gfCNCPoint1[12076] = {X 239.3673, Y 29.5319, Z -1.3333, A 0.000, B 0.000, C 0.000 }
gfCNCPoint1[12077] = {X 238.5512, Y 28.3732, Z -1.3333, A 0.000, B 0.000, C 0.000 }
gfCNCPoint1[12078] = {X 237.8897, Y 27.1197, Z -1.3333, A 0.000, B 0.000, C 0.000 }
gfCNCPoint1[12079] = {X 237.3937, Y 25.7920, Z -1.3333, A 0.000, B 0.000, C 0.000 }
gfCNCPoint1[12080] = {X 236.9799, Y 24.0072, Z -1.3333, A 0.000, B 0.000, C 0.000 }
gfCNCPoint1[12081] = {X 236.7691, Y 22.1872, Z -1.3333, A 0.000, B 0.000, C 0.000 }
gfCNCPoint1[12082] = {X 236.7640, Y 20.3550, Z -1.3333, A 0.000, B 0.000, C 0.000 }
gfCNCPoint1[12083] = {X 236.9646, Y 18.5339, Z -1.3333, A 0.000, B 0.000, C 0.000 }
gfCNCPoint1[12084] = {X 237.3683, Y 16.7468, Z -1.3333, A 0.000, B 0.000, C 0.000 }
gfCNCPoint1[12085] = {X 237.9270, Y 15.2029, Z -1.3333, A 0.000, B 0.000, C 0.000 }
gfCNCPoint1[12086] = {X 238.6980, Y 13.7534, Z -1.3333, A 0.000, B 0.000, C 0.000 }
gfCNCPoint1[12087] = {X 239.6659, Y 12.4272, Z -1.3333, A 0.000, B 0.000, C 0.000 }
gfCNCPoint1[12088] = {X 240.8112, Y 11.2509, Z -1.3333, A 0.000, B 0.000, C 0.000 }
gfCNCPoint1[12089] = {X 242.1110, Y 10.2479, Z -1.3333, A 0.000, B 0.000, C 0.000 }
gfCNCPoint1[12090] = {X 243.5394, Y 9.4385, Z -1.3333, A 0.000, B 0.000, C 0.000 }
gfCNCPoint1[12091] = {X 245.0677, Y 8.8387, Z -1.3333, A 0.000, B 0.000, C 0.000 }
gfCNCPoint1[12092] = {X 246.6654, Y 8.4605, Z -1.3333, A 0.000, B 0.000, C 0.000 }
gfCNCPoint1[12093] = {X 248.7417, Y 8.1916, Z -1.3333, A 0.000, B 0.000, C 0.000 }
gfCNCPoint1[12094] = {X 250.8339, Y 8.1119, Z -1.3333, A 0.000, B 0.000, C 0.000 }
gfCNCPoint1[12095] = {X 266.7614, Y 8.1119, Z -1.3333, A 0.000, B 0.000, C 0.000 }
gfCNCPoint1[12096] = {X 267.6634, Y 8.2203, Z -1.3333, A 0.000, B 0.000, C 0.000 }
gfCNCPoint1[12097] = {X 268.5190, Y 8.5254, Z -1.3333, A 0.000, B 0.000, C 0.000 }
gfCNCPoint1[12098] = {X 269.2860, Y 9.0122, Z -1.3333, A 0.000, B 0.000, C 0.000 }
gfCNCPoint1[12099] = {X 269.9264, Y 9.6566, Z -1.3333, A 0.000, B 0.000, C 0.000 }
gfCNCPoint1[12100] = {X 270.4084, Y 10.4266, Z -1.3333, A 0.000, B 0.000, C 0.000 }
gfCNCPoint1[12101] = {X 270.7082, Y 11.2841, Z -1.3333, A 0.000, B 0.000, C 0.000 }
gfCNCPoint1[12102] = {X 270.8110, Y 12.1867, Z -1.3333, A 0.000, B 0.000, C 0.000 }
gfCNCPoint1[12103] = {X 270.8108, Y 13.0200, Z -1.3333, A 0.000, B 0.000, C 0.000 }
gfCNCPoint1[12104] = {X 270.7022, Y 13.9141, Z -1.3333, A 0.000, B 0.000, C 0.000 }
gfCNCPoint1[12105] = {X 270.4001, Y 14.7626, Z -1.3333, A 0.000, B 0.000, C 0.000 }
gfCNCPoint1[12106] = {X 269.9191, Y 15.5241, Z -1.3333, A 0.000, B 0.000, C 0.000 }
gfCNCPoint1[12107] = {X 269.2828, Y 16.1615, Z -1.3333, A 0.000, B 0.000, C 0.000 }
gfCNCPoint1[12108] = {X 269.2827, Y 28.5937, Z -1.3333, A 0.000, B 0.000, C 0.000 }
gfCNCPoint1[12109] = {X 273.2827, Y 28.5937, Z -1.3333, A 0.000, B 0.000, C 0.000 }
gfCNCPoint1[12110] = {X 269.2027, Y 28.5937, Z -1.3333, A 0.000, B 0.000, C 0.000 }
gfCNCPoint1[12111] = {X 269.2026, Y 41.0663, Z -1.3333, A 0.000, B 0.000, C 0.000 }
gfCNCPoint1[12112] = {X 269.3416, Y 41.1781, Z -1.3333, A 0.000, B 0.000, C 0.000 }
gfCNCPoint1[12113] = {X 269.9279, Y 41.8047, Z -1.3333, A 0.000, B 0.000, C 0.000 }
gfCNCPoint1[12114] = {X 270.3671, Y 42.5419, Z -1.3333, A 0.000, B 0.000, C 0.000 }
gfCNCPoint1[12115] = {X 270.6390, Y 43.3558, Z -1.3333, A 0.000, B 0.000, C 0.000 }
gfCNCPoint1[12116] = {X 270.7310, Y 44.2089, Z -1.3333, A 0.000, B 0.000, C 0.000 }
gfCNCPoint1[12117] = {X 270.7310, Y 45.0000, Z -1.3333, A 0.000, B 0.000, C 0.000 }
gfCNCPoint1[12118] = {X 270.6307, Y 45.8901, Z -1.3333, A 0.000, B 0.000, C 0.000 }
gfCNCPoint1[12119] = {X 270.3349, Y 46.7355, Z -1.3333, A 0.000, B 0.000, C 0.000 }
gfCNCPoint1[12120] = {X 269.8584, Y 47.4940, Z -1.3333, A 0.000, B 0.000, C 0.000 }
gfCNCPoint1[12121] = {X 269.2250, Y 48.1273, Z -1.3333, A 0.000, B 0.000, C 0.000 }
gfCNCPoint1[12122] = {X 268.4666, Y 48.6039, Z -1.3333, A 0.000, B 0.000, C 0.000 }
gfCNCPoint1[12123] = {X 267.6211, Y 48.8997, Z -1.3333, A 0.000, B 0.000, C 0.000 }
gfCNCPoint1[12124] = {X 266.7310, Y 49.0000, Z -1.3333, A 0.000, B 0.000, C 0.000 }
gfCNCPoint1[12125] = {X 260.2876, Y 49.0000, Z -1.3333, A 0.000, B 0.000, C 0.000 }
gfCNCPoint1[12126] = {X 259.3975, Y 48.8997, Z -1.3333, A 0.000, B 0.000, C 0.000 }
gfCNCPoint1[12127] = {X 258.5520, Y 48.6039, Z -1.3333, A 0.000, B 0.000, C 0.000 }
gfCNCPoint1[12128] = {X 257.7936, Y 48.1273, Z -1.3333, A 0.000, B 0.000, C 0.000 }
gfCNCPoint1[12129] = {X 257.1602, Y 47.4939, Z -1.3333, A 0.000, B 0.000, C 0.000 }
gfCNCPoint1[12130] = {X 256.6837, Y 46.7355, Z -1.3333, A 0.000, B 0.000, C 0.000 }
gfCNCPoint1[12131] = {X 256.3878, Y 45.8900, Z -1.3333, A 0.000, B 0.000, C 0.000 }
gfCNCPoint1[12132] = {X 256.2876, Y 45.0000, Z -1.3333, A 0.000, B 0.000, C 0.000 }
gfCNCPoint1[12133] = {X 256.2879, Y 44.1538, Z -1.3333, A 0.000, B 0.000, C 0.000 }
gfCNCPoint1[12134] = {X 256.3986, Y 43.2730, Z -1.3333, A 0.000, B 0.000, C 0.000 }
gfCNCPoint1[12135] = {X 256.7008, Y 42.4382, Z -1.3333, A 0.000, B 0.000, C 0.000 }
gfCNCPoint1[12136] = {X 257.1796, Y 41.6907, Z -1.3333, A 0.000, B 0.000, C 0.000 }
gfCNCPoint1[12137] = {X 257.8115, Y 41.0672, Z -1.3333, A 0.000, B 0.000, C 0.000 }
gfCNCPoint1[12138] = {X 257.8115, Y 34.1538, Z -1.3333, A 0.000, B 0.000, C 0.000 }
gfCNCPoint1[12139] = {X 254.8153, Y 34.1538, Z -1.3333, A 0.000, B 0.000, C 0.000 }
gfCNCPoint1[12140] = {X 254.5724, Y 34.1511, Z -1.3333, A 0.000, B 0.000, C 0.000 }
gfCNCPoint1[12141] = {X 250.1354, Y 42.7952, Z -1.3333, A 0.000, B 0.000, C 0.000 }
gfCNCPoint1[12142] = {X 250.3285, Y 43.4904, Z -1.3333, A 0.000, B 0.000, C 0.000 }
gfCNCPoint1[12143] = {X 250.3936, Y 44.2089, Z -1.3333, A 0.000, B 0.000, C 0.000 }
gfCNCPoint1[12144] = {X 250.3936, Y 45.0000, Z -1.3333, A 0.000, B 0.000, C 0.000 }
gfCNCPoint1[12145] = {X 250.2933, Y 45.8901, Z -1.3333, A 0.000, B 0.000, C 0.000 }
gfCNCPoint1[12146] = {X 249.9974, Y 46.7355, Z -1.3333, A 0.000, B 0.000, C 0.000 }
gfCNCPoint1[12147] = {X 249.5209, Y 47.4940, Z -1.3333, A 0.000, B 0.000, C 0.000 }
gfCNCPoint1[12148] = {X 248.8875, Y 48.1273, Z -1.3333, A 0.000, B 0.000, C 0.000 }
gfCNCPoint1[12149] = {X 248.1291, Y 48.6039, Z -1.3333, A 0.000, B 0.000, C 0.000 }
gfCNCPoint1[12150] = {X 247.2836, Y 48.8997, Z -1.3333, A 0.000, B 0.000, C 0.000 }
gfCNCPoint1[12151] = {X 246.3936, Y 49.0000, Z -1.3333, A 0.000, B 0.000, C 0.000 }
gfCNCPoint1[12152] = {X 239.8075, Y 49.0000, Z -1.3333, A 0.000, B 0.000, C 0.000 }
gfCNCPoint1[12153] = {X 238.9174, Y 48.8997, Z -1.3333, A 0.000, B 0.000, C 0.000 }
gfCNCPoint1[12154] = {X 238.0720, Y 48.6039, Z -1.3333, A 0.000, B 0.000, C 0.000 }
gfCNCPoint1[12155] = {X 237.3135, Y 48.1273, Z -1.3333, A 0.000, B 0.000, C 0.000 }
gfCNCPoint1[12156] = {X 236.6802, Y 47.4940, Z -1.3333, A 0.000, B 0.000, C 0.000 }
gfCNCPoint1[12157] = {X 236.2036, Y 46.7355, Z -1.3333, A 0.000, B 0.000, C 0.000 }
gfCNCPoint1[12158] = {X 235.9078, Y 45.8901, Z -1.3333, A 0.000, B 0.000, C 0.000 }
gfCNCPoint1[12159] = {X 235.8075, Y 45.0000, Z -1.3333, A 0.000, B 0.000, C 0.000 }
gfCNCPoint1[12160] = {X 235.8079, Y 44.1538, Z -1.3333, A 0.000, B 0.000, C 0.000 }
gfCNCPoint1[12161] = {X 235.9027, Y 43.3414, Z -1.3333, A 0.000, B 0.000, C 0.000 }
gfCNCPoint1[12162] = {X 236.1607, Y 42.5654, Z -1.3333, A 0.000, B 0.000, C 0.000 }
gfCNCPoint1[12163] = {X 236.5712, Y 41.8580, Z -1.3333, A 0.000, B 0.000, C 0.000 }
gfCNCPoint1[12164] = {X 237.1169, Y 41.2489, Z -1.3333, A 0.000, B 0.000, C 0.000 }
gfCNCPoint1[12165] = {X 237.7752, Y 40.7635, Z -1.3333, A 0.000, B 0.000, C 0.000 }
gfCNCPoint1[12166] = {X 238.5184, Y 40.4222, Z -1.3333, A 0.000, B 0.000, C 0.000 }
gfCNCPoint1[12167] = {X 242.7051, Y 32.2271, Z -1.3333, A 0.000, B 0.000, C 0.000 }
gfCNCPoint1[12168] = {X 241.5071, Y 31.4650, Z -1.3333, A 0.000, B 0.000, C 0.000 }
gfCNCPoint1[12169] = {X 240.4173, Y 30.5548, Z -1.3333, A 0.000, B 0.000, C 0.000 }
gfCNCPoint1[12170] = {X 239.4538, Y 29.5118, Z -1.3333, A 0.000, B 0.000, C 0.000 }
gfCNCPoint1[12171] = {X 238.6328, Y 28.3533, Z -1.3333, A 0.000, B 0.000, C 0.000 }
gfCNCPoint1[12172] = {X 237.9679, Y 27.0987, Z -1.3333, A 0.000, B 0.000, C 0.000 }
gfCNCPoint1[12173] = {X 237.4702, Y 25.7689, Z -1.3333, A 0.000, B 0.000, C 0.000 }
gfCNCPoint1[12174] = {X 237.0586, Y 23.9929, Z -1.3333, A 0.000, B 0.000, C 0.000 }
gfCNCPoint1[12175] = {X 236.8490, Y 22.1820, Z -1.3333, A 0.000, B 0.000, C 0.000 }
gfCNCPoint1[12176] = {X 236.8439, Y 20.3590, Z -1.3333, A 0.000, B 0.000, C 0.000 }
gfCNCPoint1[12177] = {X 237.0435, Y 18.5469, Z -1.3333, A 0.000, B 0.000, C 0.000 }
gfCNCPoint1[12178] = {X 237.4452, Y 16.7687, Z -1.3333, A 0.000, B 0.000, C 0.000 }
gfCNCPoint1[12179] = {X 238.0001, Y 15.2355, Z -1.3333, A 0.000, B 0.000, C 0.000 }
gfCNCPoint1[12180] = {X 238.7658, Y 13.7959, Z -1.3333, A 0.000, B 0.000, C 0.000 }
gfCNCPoint1[12181] = {X 239.7270, Y 12.4788, Z -1.3333, A 0.000, B 0.000, C 0.000 }
gfCNCPoint1[12182] = {X 240.8645, Y 11.3105, Z -1.3333, A 0.000, B 0.000, C 0.000 }
gfCNCPoint1[12183] = {X 242.1555, Y 10.3144, Z -1.3333, A 0.000, B 0.000, C 0.000 }
gfCNCPoint1[12184] = {X 243.5741, Y 9.5105, Z -1.3333, A 0.000, B 0.000, C 0.000 }
gfCNCPoint1[12185] = {X 245.0920, Y 8.9149, Z -1.3333, A 0.000, B 0.000, C 0.000 }
gfCNCPoint1[12186] = {X 246.6787, Y 8.5394, Z -1.3333, A 0.000, B 0.000, C 0.000 }
gfCNCPoint1[12187] = {X 248.7483, Y 8.2713, Z -1.3333, A 0.000, B 0.000, C 0.000 }
gfCNCPoint1[12188] = {X 250.8336, Y 8.1919, Z -1.3333, A 0.000, B 0.000, C 0.000 }
gfCNCPoint1[12189] = {X 266.7608, Y 8.1919, Z -1.3333, A 0.000, B 0.000, C 0.000 }
gfCNCPoint1[12190] = {X 267.6450, Y 8.2982, Z -1.3333, A 0.000, B 0.000, C 0.000 }
gfCNCPoint1[12191] = {X 268.4839, Y 8.5973, Z -1.3333, A 0.000, B 0.000, C 0.000 }
gfCNCPoint1[12192] = {X 269.2359, Y 9.0746, Z -1.3333, A 0.000, B 0.000, C 0.000 }
gfCNCPoint1[12193] = {X 269.8637, Y 9.7063, Z -1.3333, A 0.000, B 0.000, C 0.000 }
gfCNCPoint1[12194] = {X 270.3363, Y 10.4612, Z -1.3333, A 0.000, B 0.000, C 0.000 }
gfCNCPoint1[12195] = {X 270.6303, Y 11.3020, Z -1.3333, A 0.000, B 0.000, C 0.000 }
gfCNCPoint1[12196] = {X 270.7310, Y 12.1869, Z -1.3333, A 0.000, B 0.000, C 0.000 }
gfCNCPoint1[12197] = {X 270.7308, Y 13.0192, Z -1.3333, A 0.000, B 0.000, C 0.000 }
gfCNCPoint1[12198] = {X 270.6221, Y 13.9051, Z -1.3333, A 0.000, B 0.000, C 0.000 }
gfCNCPoint1[12199] = {X 270.3197, Y 14.7448, Z -1.3333, A 0.000, B 0.000, C 0.000 }
gfCNCPoint1[12200] = {X 269.8386, Y 15.4965, Z -1.3333, A 0.000, B 0.000, C 0.000 }
gfCNCPoint1[12201] = {X 269.2028, Y 16.1229, Z -1.3333, A 0.000, B 0.000, C 0.000 }
gfCNCPoint1[12202] = {X 269.2027, Y 28.5937, Z -1.3333, A 0.000, B 0.000, C 0.000 }
gfCNCPoint1[12203] = {X 273.2827, Y 28.5937, Z -1.3333, A 0.000, B 0.000, C 0.000 }
gfCNCPoint1[12204] = {X 273.2827, Y 28.5937, Z 1.6667, A 0.000, B 0.000, C 0.000 }
gfCNCPoint1[12205] = {X 273.2827, Y 28.5937, Z 11.0000, A 0.000, B 0.000, C 0.000 }
gfCNCPoint1[12206] = {X 277.7463, Y 28.5933, Z 11.0000, A 0.000, B 0.000, C 0.000 }
gfCNCPoint1[12207] = {X 277.7463, Y 28.5933, Z 1.6667, A 0.000, B 0.000, C 0.000 }
gfCNCPoint1[12208] = {X 277.7463, Y 28.5933, Z -1.3333, A 0.000, B 0.000, C 0.000 }
gfCNCPoint1[12209] = {X 281.8263, Y 28.5932, Z -1.3333, A 0.000, B 0.000, C 0.000 }
gfCNCPoint1[12210] = {X 281.8261, Y 16.2749, Z -1.3333, A 0.000, B 0.000, C 0.000 }
gfCNCPoint1[12211] = {X 281.1872, Y 15.6037, Z -1.3333, A 0.000, B 0.000, C 0.000 }
gfCNCPoint1[12212] = {X 280.7062, Y 14.8118, Z -1.3333, A 0.000, B 0.000, C 0.000 }
gfCNCPoint1[12213] = {X 280.4051, Y 13.9354, Z -1.3333, A 0.000, B 0.000, C 0.000 }
gfCNCPoint1[12214] = {X 280.2978, Y 13.0150, Z -1.3333, A 0.000, B 0.000, C 0.000 }
gfCNCPoint1[12215] = {X 280.2977, Y 12.1868, Z -1.3333, A 0.000, B 0.000, C 0.000 }
gfCNCPoint1[12216] = {X 280.4060, Y 11.2255, Z -1.3333, A 0.000, B 0.000, C 0.000 }
gfCNCPoint1[12217] = {X 280.7255, Y 10.3124, Z -1.3333, A 0.000, B 0.000, C 0.000 }
gfCNCPoint1[12218] = {X 281.2402, Y 9.4933, Z -1.3333, A 0.000, B 0.000, C 0.000 }
gfCNCPoint1[12219] = {X 281.9242, Y 8.8093, Z -1.3333, A 0.000, B 0.000, C 0.000 }
gfCNCPoint1[12220] = {X 282.7433, Y 8.2946, Z -1.3333, A 0.000, B 0.000, C 0.000 }
gfCNCPoint1[12221] = {X 283.6564, Y 7.9751, Z -1.3333, A 0.000, B 0.000, C 0.000 }
gfCNCPoint1[12222] = {X 284.6177, Y 7.8668, Z -1.3333, A 0.000, B 0.000, C 0.000 }
gfCNCPoint1[12223] = {X 291.0611, Y 7.8668, Z -1.3333, A 0.000, B 0.000, C 0.000 }
gfCNCPoint1[12224] = {X 292.0224, Y 7.9751, Z -1.3333, A 0.000, B 0.000, C 0.000 }
gfCNCPoint1[12225] = {X 292.9355, Y 8.2946, Z -1.3333, A 0.000, B 0.000, C 0.000 }
gfCNCPoint1[12226] = {X 293.7546, Y 8.8093, Z -1.3333, A 0.000, B 0.000, C 0.000 }
gfCNCPoint1[12227] = {X 294.4386, Y 9.4933, Z -1.3333, A 0.000, B 0.000, C 0.000 }
gfCNCPoint1[12228] = {X 294.9533, Y 10.3124, Z -1.3333, A 0.000, B 0.000, C 0.000 }
gfCNCPoint1[12229] = {X 295.2728, Y 11.2255, Z -1.3333, A 0.000, B 0.000, C 0.000 }
gfCNCPoint1[12230] = {X 295.3811, Y 12.1868, Z -1.3333, A 0.000, B 0.000, C 0.000 }
gfCNCPoint1[12231] = {X 295.3811, Y 12.9781, Z -1.3333, A 0.000, B 0.000, C 0.000 }
gfCNCPoint1[12232] = {X 295.2797, Y 13.9084, Z -1.3333, A 0.000, B 0.000, C 0.000 }
gfCNCPoint1[12233] = {X 294.9802, Y 14.7950, Z -1.3333, A 0.000, B 0.000, C 0.000 }
gfCNCPoint1[12234] = {X 294.4969, Y 15.5963, Z -1.3333, A 0.000, B 0.000, C 0.000 }
gfCNCPoint1[12235] = {X 293.8524, Y 16.2748, Z -1.3333, A 0.000, B 0.000, C 0.000 }
gfCNCPoint1[12236] = {X 293.8537, Y 22.1965, Z -1.3333, A 0.000, B 0.000, C 0.000 }
gfCNCPoint1[12237] = {X 302.7601, Y 22.1965, Z -1.3333, A 0.000, B 0.000, C 0.000 }
gfCNCPoint1[12238] = {X 302.7648, Y 16.2784, Z -1.3333, A 0.000, B 0.000, C 0.000 }
gfCNCPoint1[12239] = {X 302.1245, Y 15.6073, Z -1.3333, A 0.000, B 0.000, C 0.000 }
gfCNCPoint1[12240] = {X 301.6422, Y 14.8149, Z -1.3333, A 0.000, B 0.000, C 0.000 }
gfCNCPoint1[12241] = {X 301.3402, Y 13.9378, Z -1.3333, A 0.000, B 0.000, C 0.000 }
gfCNCPoint1[12242] = {X 301.2324, Y 13.0165, Z -1.3333, A 0.000, B 0.000, C 0.000 }
gfCNCPoint1[12243] = {X 301.2323, Y 12.1868, Z -1.3333, A 0.000, B 0.000, C 0.000 }
gfCNCPoint1[12244] = {X 301.3406, Y 11.2255, Z -1.3333, A 0.000, B 0.000, C 0.000 }
gfCNCPoint1[12245] = {X 301.6601, Y 10.3124, Z -1.3333, A 0.000, B 0.000, C 0.000 }
gfCNCPoint1[12246] = {X 302.1747, Y 9.4933, Z -1.3333, A 0.000, B 0.000, C 0.000 }
gfCNCPoint1[12247] = {X 302.8588, Y 8.8093, Z -1.3333, A 0.000, B 0.000, C 0.000 }
gfCNCPoint1[12248] = {X 303.6779, Y 8.2946, Z -1.3333, A 0.000, B 0.000, C 0.000 }
gfCNCPoint1[12249] = {X 304.5910, Y 7.9751, Z -1.3333, A 0.000, B 0.000, C 0.000 }
gfCNCPoint1[12250] = {X 305.5523, Y 7.8668, Z -1.3333, A 0.000, B 0.000, C 0.000 }
gfCNCPoint1[12251] = {X 311.9957, Y 7.8668, Z -1.3333, A 0.000, B 0.000, C 0.000 }
gfCNCPoint1[12252] = {X 312.9570, Y 7.9751, Z -1.3333, A 0.000, B 0.000, C 0.000 }
gfCNCPoint1[12253] = {X 313.8701, Y 8.2946, Z -1.3333, A 0.000, B 0.000, C 0.000 }
gfCNCPoint1[12254] = {X 314.6892, Y 8.8093, Z -1.3333, A 0.000, B 0.000, C 0.000 }
gfCNCPoint1[12255] = {X 315.3732, Y 9.4933, Z -1.3333, A 0.000, B 0.000, C 0.000 }
gfCNCPoint1[12256] = {X 315.8879, Y 10.3124, Z -1.3333, A 0.000, B 0.000, C 0.000 }
gfCNCPoint1[12257] = {X 316.2074, Y 11.2255, Z -1.3333, A 0.000, B 0.000, C 0.000 }
gfCNCPoint1[12258] = {X 316.3157, Y 12.1868, Z -1.3333, A 0.000, B 0.000, C 0.000 }
gfCNCPoint1[12259] = {X 316.3157, Y 12.9781, Z -1.3333, A 0.000, B 0.000, C 0.000 }
gfCNCPoint1[12260] = {X 316.2143, Y 13.9085, Z -1.3333, A 0.000, B 0.000, C 0.000 }
gfCNCPoint1[12261] = {X 315.9150, Y 14.7951, Z -1.3333, A 0.000, B 0.000, C 0.000 }
gfCNCPoint1[12262] = {X 315.4317, Y 15.5965, Z -1.3333, A 0.000, B 0.000, C 0.000 }
gfCNCPoint1[12263] = {X 314.7871, Y 16.2750, Z -1.3333, A 0.000, B 0.000, C 0.000 }
gfCNCPoint1[12264] = {X 314.7869, Y 40.9116, Z -1.3333, A 0.000, B 0.000, C 0.000 }
gfCNCPoint1[12265] = {X 315.4259, Y 41.5826, Z -1.3333, A 0.000, B 0.000, C 0.000 }
gfCNCPoint1[12266] = {X 315.9070, Y 42.3746, Z -1.3333, A 0.000, B 0.000, C 0.000 }
gfCNCPoint1[12267] = {X 316.2082, Y 43.2509, Z -1.3333, A 0.000, B 0.000, C 0.000 }
gfCNCPoint1[12268] = {X 316.3156, Y 44.1713, Z -1.3333, A 0.000, B 0.000, C 0.000 }
gfCNCPoint1[12269] = {X 316.3157, Y 45.0000, Z -1.3333, A 0.000, B 0.000, C 0.000 }
gfCNCPoint1[12270] = {X 316.2074, Y 45.9613, Z -1.3333, A 0.000, B 0.000, C 0.000 }
gfCNCPoint1[12271] = {X 315.8879, Y 46.8744, Z -1.3333, A 0.000, B 0.000, C 0.000 }
gfCNCPoint1[12272] = {X 315.3732, Y 47.6935, Z -1.3333, A 0.000, B 0.000, C 0.000 }
gfCNCPoint1[12273] = {X 314.6892, Y 48.3775, Z -1.3333, A 0.000, B 0.000, C 0.000 }
gfCNCPoint1[12274] = {X 313.8701, Y 48.8922, Z -1.3333, A 0.000, B 0.000, C 0.000 }
gfCNCPoint1[12275] = {X 312.9570, Y 49.2117, Z -1.3333, A 0.000, B 0.000, C 0.000 }
gfCNCPoint1[12276] = {X 311.9957, Y 49.3200, Z -1.3333, A 0.000, B 0.000, C 0.000 }
gfCNCPoint1[12277] = {X 305.5523, Y 49.3200, Z -1.3333, A 0.000, B 0.000, C 0.000 }
gfCNCPoint1[12278] = {X 304.5958, Y 49.2128, Z -1.3333, A 0.000, B 0.000, C 0.000 }
gfCNCPoint1[12279] = {X 303.6868, Y 48.8965, Z -1.3333, A 0.000, B 0.000, C 0.000 }
gfCNCPoint1[12280] = {X 302.8704, Y 48.3868, Z -1.3333, A 0.000, B 0.000, C 0.000 }
gfCNCPoint1[12281] = {X 302.1872, Y 47.7090, Z -1.3333, A 0.000, B 0.000, C 0.000 }
gfCNCPoint1[12282] = {X 301.6709, Y 46.8967, Z -1.3333, A 0.000, B 0.000, C 0.000 }
gfCNCPoint1[12283] = {X 301.3473, Y 45.9903, Z -1.3333, A 0.000, B 0.000, C 0.000 }
gfCNCPoint1[12284] = {X 301.2324, Y 45.0348, Z -1.3333, A 0.000, B 0.000, C 0.000 }
gfCNCPoint1[12285] = {X 301.2324, Y 44.2010, Z -1.3333, A 0.000, B 0.000, C 0.000 }
gfCNCPoint1[12286] = {X 301.3506, Y 43.2650, Z -1.3333, A 0.000, B 0.000, C 0.000 }
gfCNCPoint1[12287] = {X 301.6542, Y 42.3717, Z -1.3333, A 0.000, B 0.000, C 0.000 }
gfCNCPoint1[12288] = {X 302.1308, Y 41.5575, Z -1.3333, A 0.000, B 0.000, C 0.000 }
gfCNCPoint1[12289] = {X 302.7611, Y 40.8554, Z -1.3333, A 0.000, B 0.000, C 0.000 }
gfCNCPoint1[12290] = {X 302.7611, Y 34.0343, Z -1.3333, A 0.000, B 0.000, C 0.000 }
gfCNCPoint1[12291] = {X 293.8535, Y 34.0343, Z -1.3333, A 0.000, B 0.000, C 0.000 }
gfCNCPoint1[12292] = {X 293.8525, Y 40.9029, Z -1.3333, A 0.000, B 0.000, C 0.000 }
gfCNCPoint1[12293] = {X 294.4915, Y 41.5869, Z -1.3333, A 0.000, B 0.000, C 0.000 }
gfCNCPoint1[12294] = {X 294.9723, Y 42.3901, Z -1.3333, A 0.000, B 0.000, C 0.000 }
gfCNCPoint1[12295] = {X 295.2733, Y 43.2764, Z -1.3333, A 0.000, B 0.000, C 0.000 }
gfCNCPoint1[12296] = {X 295.3811, Y 44.2063, Z -1.3333, A 0.000, B 0.000, C 0.000 }
gfCNCPoint1[12297] = {X 295.3811, Y 45.0000, Z -1.3333, A 0.000, B 0.000, C 0.000 }
gfCNCPoint1[12298] = {X 295.2728, Y 45.9613, Z -1.3333, A 0.000, B 0.000, C 0.000 }
gfCNCPoint1[12299] = {X 294.9533, Y 46.8744, Z -1.3333, A 0.000, B 0.000, C 0.000 }
gfCNCPoint1[12300] = {X 294.4386, Y 47.6935, Z -1.3333, A 0.000, B 0.000, C 0.000 }
gfCNCPoint1[12301] = {X 293.7546, Y 48.3775, Z -1.3333, A 0.000, B 0.000, C 0.000 }
gfCNCPoint1[12302] = {X 292.9355, Y 48.8922, Z -1.3333, A 0.000, B 0.000, C 0.000 }
gfCNCPoint1[12303] = {X 292.0224, Y 49.2117, Z -1.3333, A 0.000, B 0.000, C 0.000 }
gfCNCPoint1[12304] = {X 291.0611, Y 49.3200, Z -1.3333, A 0.000, B 0.000, C 0.000 }
gfCNCPoint1[12305] = {X 284.6177, Y 49.3200, Z -1.3333, A 0.000, B 0.000, C 0.000 }
gfCNCPoint1[12306] = {X 283.6613, Y 49.2128, Z -1.3333, A 0.000, B 0.000, C 0.000 }
gfCNCPoint1[12307] = {X 282.7524, Y 48.8965, Z -1.3333, A 0.000, B 0.000, C 0.000 }
gfCNCPoint1[12308] = {X 281.9360, Y 48.3869, Z -1.3333, A 0.000, B 0.000, C 0.000 }
gfCNCPoint1[12309] = {X 281.2527, Y 47.7092, Z -1.3333, A 0.000, B 0.000, C 0.000 }
gfCNCPoint1[12310] = {X 280.7365, Y 46.8970, Z -1.3333, A 0.000, B 0.000, C 0.000 }
gfCNCPoint1[12311] = {X 280.4128, Y 45.9907, Z -1.3333, A 0.000, B 0.000, C 0.000 }
gfCNCPoint1[12312] = {X 280.2978, Y 45.0352, Z -1.3333, A 0.000, B 0.000, C 0.000 }
gfCNCPoint1[12313] = {X 280.2977, Y 44.2069, Z -1.3333, A 0.000, B 0.000, C 0.000 }
gfCNCPoint1[12314] = {X 280.4033, Y 43.2781, Z -1.3333, A 0.000, B 0.000, C 0.000 }
gfCNCPoint1[12315] = {X 280.7038, Y 42.3930, Z -1.3333, A 0.000, B 0.000, C 0.000 }
gfCNCPoint1[12316] = {X 281.1856, Y 41.5919, Z -1.3333, A 0.000, B 0.000, C 0.000 }
gfCNCPoint1[12317] = {X 281.8265, Y 40.9115, Z -1.3333, A 0.000, B 0.000, C 0.000 }
gfCNCPoint1[12318] = {X 281.8263, Y 28.5932, Z -1.3333, A 0.000, B 0.000, C 0.000 }
gfCNCPoint1[12319] = {X 277.8263, Y 28.5933, Z -1.3333, A 0.000, B 0.000, C 0.000 }
gfCNCPoint1[12320] = {X 281.9063, Y 28.5932, Z -1.3333, A 0.000, B 0.000, C 0.000 }
gfCNCPoint1[12321] = {X 281.9061, Y 16.2376, Z -1.3333, A 0.000, B 0.000, C 0.000 }
gfCNCPoint1[12322] = {X 281.2677, Y 15.5771, Z -1.3333, A 0.000, B 0.000, C 0.000 }
gfCNCPoint1[12323] = {X 280.7865, Y 14.7945, Z -1.3333, A 0.000, B 0.000, C 0.000 }
gfCNCPoint1[12324] = {X 280.4852, Y 13.9267, Z -1.3333, A 0.000, B 0.000, C 0.000 }
gfCNCPoint1[12325] = {X 280.3778, Y 13.0143, Z -1.3333, A 0.000, B 0.000, C 0.000 }
gfCNCPoint1[12326] = {X 280.3777, Y 12.1868, Z -1.3333, A 0.000, B 0.000, C 0.000 }
gfCNCPoint1[12327] = {X 280.4840, Y 11.2433, Z -1.3333, A 0.000, B 0.000, C 0.000 }
gfCNCPoint1[12328] = {X 280.7976, Y 10.3472, Z -1.3333, A 0.000, B 0.000, C 0.000 }
gfCNCPoint1[12329] = {X 281.3027, Y 9.5432, Z -1.3333, A 0.000, B 0.000, C 0.000 }
gfCNCPoint1[12330] = {X 281.9741, Y 8.8719, Z -1.3333, A 0.000, B 0.000, C 0.000 }
gfCNCPoint1[12331] = {X 282.7780, Y 8.3667, Z -1.3333, A 0.000, B 0.000, C 0.000 }
gfCNCPoint1[12332] = {X 283.6742, Y 8.0531, Z -1.3333, A 0.000, B 0.000, C 0.000 }
gfCNCPoint1[12333] = {X 284.6177, Y 7.9468, Z -1.3333, A 0.000, B 0.000, C 0.000 }
gfCNCPoint1[12334] = {X 291.0611, Y 7.9468, Z -1.3333, A 0.000, B 0.000, C 0.000 }
gfCNCPoint1[12335] = {X 292.0046, Y 8.0531, Z -1.3333, A 0.000, B 0.000, C 0.000 }
gfCNCPoint1[12336] = {X 292.9008, Y 8.3667, Z -1.3333, A 0.000, B 0.000, C 0.000 }
gfCNCPoint1[12337] = {X 293.7047, Y 8.8718, Z -1.3333, A 0.000, B 0.000, C 0.000 }
gfCNCPoint1[12338] = {X 294.3761, Y 9.5432, Z -1.3333, A 0.000, B 0.000, C 0.000 }
gfCNCPoint1[12339] = {X 294.8812, Y 10.3471, Z -1.3333, A 0.000, B 0.000, C 0.000 }
gfCNCPoint1[12340] = {X 295.1948, Y 11.2433, Z -1.3333, A 0.000, B 0.000, C 0.000 }
gfCNCPoint1[12341] = {X 295.3011, Y 12.1868, Z -1.3333, A 0.000, B 0.000, C 0.000 }
gfCNCPoint1[12342] = {X 295.3011, Y 12.9781, Z -1.3333, A 0.000, B 0.000, C 0.000 }
gfCNCPoint1[12343] = {X 295.1995, Y 13.9002, Z -1.3333, A 0.000, B 0.000, C 0.000 }
gfCNCPoint1[12344] = {X 294.8999, Y 14.7781, Z -1.3333, A 0.000, B 0.000, C 0.000 }
gfCNCPoint1[12345] = {X 294.4164, Y 15.5698, Z -1.3333, A 0.000, B 0.000, C 0.000 }
gfCNCPoint1[12346] = {X 293.7724, Y 16.2375, Z -1.3333, A 0.000, B 0.000, C 0.000 }
gfCNCPoint1[12347] = {X 293.7738, Y 22.2765, Z -1.3333, A 0.000, B 0.000, C 0.000 }
gfCNCPoint1[12348] = {X 302.8400, Y 22.2765, Z -1.3333, A 0.000, B 0.000, C 0.000 }
gfCNCPoint1[12349] = {X 302.8449, Y 16.2411, Z -1.3333, A 0.000, B 0.000, C 0.000 }
gfCNCPoint1[12350] = {X 302.2050, Y 15.5806, Z -1.3333, A 0.000, B 0.000, C 0.000 }
gfCNCPoint1[12351] = {X 301.7226, Y 14.7976, Z -1.3333, A 0.000, B 0.000, C 0.000 }
gfCNCPoint1[12352] = {X 301.4203, Y 13.9291, Z -1.3333, A 0.000, B 0.000, C 0.000 }
gfCNCPoint1[12353] = {X 301.3124, Y 13.0158, Z -1.3333, A 0.000, B 0.000, C 0.000 }
gfCNCPoint1[12354] = {X 301.3123, Y 12.1868, Z -1.3333, A 0.000, B 0.000, C 0.000 }
gfCNCPoint1[12355] = {X 301.4186, Y 11.2433, Z -1.3333, A 0.000, B 0.000, C 0.000 }
gfCNCPoint1[12356] = {X 301.7321, Y 10.3471, Z -1.3333, A 0.000, B 0.000, C 0.000 }
gfCNCPoint1[12357] = {X 302.2373, Y 9.5432, Z -1.3333, A 0.000, B 0.000, C 0.000 }
gfCNCPoint1[12358] = {X 302.9087, Y 8.8718, Z -1.3333, A 0.000, B 0.000, C 0.000 }
gfCNCPoint1[12359] = {X 303.7126, Y 8.3667, Z -1.3333, A 0.000, B 0.000, C 0.000 }
gfCNCPoint1[12360] = {X 304.6088, Y 8.0531, Z -1.3333, A 0.000, B 0.000, C 0.000 }
gfCNCPoint1[12361] = {X 305.5523, Y 7.9468, Z -1.3333, A 0.000, B 0.000, C 0.000 }
gfCNCPoint1[12362] = {X 311.9957, Y 7.9468, Z -1.3333, A 0.000, B 0.000, C 0.000 }
gfCNCPoint1[12363] = {X 312.9392, Y 8.0531, Z -1.3333, A 0.000, B 0.000, C 0.000 }
gfCNCPoint1[12364] = {X 313.8354, Y 8.3667, Z -1.3333, A 0.000, B 0.000, C 0.000 }
gfCNCPoint1[12365] = {X 314.6393, Y 8.8718, Z -1.3333, A 0.000, B 0.000, C 0.000 }
gfCNCPoint1[12366] = {X 315.3107, Y 9.5432, Z -1.3333, A 0.000, B 0.000, C 0.000 }
gfCNCPoint1[12367] = {X 315.8158, Y 10.3471, Z -1.3333, A 0.000, B 0.000, C 0.000 }
gfCNCPoint1[12368] = {X 316.1294, Y 11.2433, Z -1.3333, A 0.000, B 0.000, C 0.000 }
gfCNCPoint1[12369] = {X 316.2357, Y 12.1868, Z -1.3333, A 0.000, B 0.000, C 0.000 }
gfCNCPoint1[12370] = {X 316.2357, Y 12.9781, Z -1.3333, A 0.000, B 0.000, C 0.000 }
gfCNCPoint1[12371] = {X 316.1342, Y 13.9003, Z -1.3333, A 0.000, B 0.000, C 0.000 }
gfCNCPoint1[12372] = {X 315.8346, Y 14.7782, Z -1.3333, A 0.000, B 0.000, C 0.000 }
gfCNCPoint1[12373] = {X 315.3512, Y 15.5700, Z -1.3333, A 0.000, B 0.000, C 0.000 }
gfCNCPoint1[12374] = {X 314.7071, Y 16.2377, Z -1.3333, A 0.000, B 0.000, C 0.000 }
gfCNCPoint1[12375] = {X 314.7069, Y 40.9503, Z -1.3333, A 0.000, B 0.000, C 0.000 }
gfCNCPoint1[12376] = {X 314.7352, Y 40.9726, Z -1.3333, A 0.000, B 0.000, C 0.000 }
gfCNCPoint1[12377] = {X 315.3623, Y 41.6313, Z -1.3333, A 0.000, B 0.000, C 0.000 }
gfCNCPoint1[12378] = {X 315.8346, Y 42.4085, Z -1.3333, A 0.000, B 0.000, C 0.000 }
gfCNCPoint1[12379] = {X 316.1302, Y 43.2686, Z -1.3333, A 0.000, B 0.000, C 0.000 }
gfCNCPoint1[12380] = {X 316.2356, Y 44.1720, Z -1.3333, A 0.000, B 0.000, C 0.000 }
gfCNCPoint1[12381] = {X 316.2357, Y 45.0000, Z -1.3333, A 0.000, B 0.000, C 0.000 }
gfCNCPoint1[12382] = {X 316.1294, Y 45.9435, Z -1.3333, A 0.000, B 0.000, C 0.000 }
gfCNCPoint1[12383] = {X 315.8158, Y 46.8397, Z -1.3333, A 0.000, B 0.000, C 0.000 }
gfCNCPoint1[12384] = {X 315.3107, Y 47.6436, Z -1.3333, A 0.000, B 0.000, C 0.000 }
gfCNCPoint1[12385] = {X 314.6393, Y 48.3150, Z -1.3333, A 0.000, B 0.000, C 0.000 }
gfCNCPoint1[12386] = {X 313.8354, Y 48.8201, Z -1.3333, A 0.000, B 0.000, C 0.000 }
gfCNCPoint1[12387] = {X 312.9392, Y 49.1337, Z -1.3333, A 0.000, B 0.000, C 0.000 }
gfCNCPoint1[12388] = {X 311.9957, Y 49.2400, Z -1.3333, A 0.000, B 0.000, C 0.000 }
gfCNCPoint1[12389] = {X 305.5523, Y 49.2400, Z -1.3333, A 0.000, B 0.000, C 0.000 }
gfCNCPoint1[12390] = {X 304.6135, Y 49.1348, Z -1.3333, A 0.000, B 0.000, C 0.000 }
gfCNCPoint1[12391] = {X 303.7214, Y 48.8243, Z -1.3333, A 0.000, B 0.000, C 0.000 }
gfCNCPoint1[12392] = {X 302.9201, Y 48.3241, Z -1.3333, A 0.000, B 0.000, C 0.000 }
gfCNCPoint1[12393] = {X 302.2495, Y 47.6588, Z -1.3333, A 0.000, B 0.000, C 0.000 }
gfCNCPoint1[12394] = {X 301.7428, Y 46.8616, Z -1.3333, A 0.000, B 0.000, C 0.000 }
gfCNCPoint1[12395] = {X 301.4252, Y 45.9720, Z -1.3333, A 0.000, B 0.000, C 0.000 }
gfCNCPoint1[12396] = {X 301.3124, Y 45.0341, Z -1.3333, A 0.000, B 0.000, C 0.000 }
gfCNCPoint1[12397] = {X 301.3123, Y 44.2030, Z -1.3333, A 0.000, B 0.000, C 0.000 }
gfCNCPoint1[12398] = {X 301.4305, Y 43.2744, Z -1.3333, A 0.000, B 0.000, C 0.000 }
gfCNCPoint1[12399] = {X 301.7343, Y 42.3889, Z -1.3333, A 0.000, B 0.000, C 0.000 }
gfCNCPoint1[12400] = {X 302.2111, Y 41.5833, Z -1.3333, A 0.000, B 0.000, C 0.000 }
gfCNCPoint1[12401] = {X 302.8411, Y 40.8909, Z -1.3333, A 0.000, B 0.000, C 0.000 }
gfCNCPoint1[12402] = {X 302.8411, Y 33.9543, Z -1.3333, A 0.000, B 0.000, C 0.000 }
gfCNCPoint1[12403] = {X 293.7735, Y 33.9543, Z -1.3333, A 0.000, B 0.000, C 0.000 }
gfCNCPoint1[12404] = {X 293.7724, Y 40.9397, Z -1.3333, A 0.000, B 0.000, C 0.000 }
gfCNCPoint1[12405] = {X 294.4111, Y 41.6133, Z -1.3333, A 0.000, B 0.000, C 0.000 }
gfCNCPoint1[12406] = {X 294.8920, Y 42.4072, Z -1.3333, A 0.000, B 0.000, C 0.000 }
gfCNCPoint1[12407] = {X 295.1933, Y 43.2851, Z -1.3333, A 0.000, B 0.000, C 0.000 }
gfCNCPoint1[12408] = {X 295.3011, Y 44.2070, Z -1.3333, A 0.000, B 0.000, C 0.000 }
gfCNCPoint1[12409] = {X 295.3011, Y 45.0000, Z -1.3333, A 0.000, B 0.000, C 0.000 }
gfCNCPoint1[12410] = {X 295.1948, Y 45.9435, Z -1.3333, A 0.000, B 0.000, C 0.000 }
gfCNCPoint1[12411] = {X 294.8812, Y 46.8397, Z -1.3333, A 0.000, B 0.000, C 0.000 }
gfCNCPoint1[12412] = {X 294.3761, Y 47.6436, Z -1.3333, A 0.000, B 0.000, C 0.000 }
gfCNCPoint1[12413] = {X 293.7047, Y 48.3150, Z -1.3333, A 0.000, B 0.000, C 0.000 }
gfCNCPoint1[12414] = {X 292.9008, Y 48.8201, Z -1.3333, A 0.000, B 0.000, C 0.000 }
gfCNCPoint1[12415] = {X 292.0046, Y 49.1337, Z -1.3333, A 0.000, B 0.000, C 0.000 }
gfCNCPoint1[12416] = {X 291.0611, Y 49.2400, Z -1.3333, A 0.000, B 0.000, C 0.000 }
gfCNCPoint1[12417] = {X 284.6177, Y 49.2400, Z -1.3333, A 0.000, B 0.000, C 0.000 }
gfCNCPoint1[12418] = {X 283.6790, Y 49.1348, Z -1.3333, A 0.000, B 0.000, C 0.000 }
gfCNCPoint1[12419] = {X 282.7869, Y 48.8244, Z -1.3333, A 0.000, B 0.000, C 0.000 }
gfCNCPoint1[12420] = {X 281.9857, Y 48.3242, Z -1.3333, A 0.000, B 0.000, C 0.000 }
gfCNCPoint1[12421] = {X 281.3150, Y 47.6590, Z -1.3333, A 0.000, B 0.000, C 0.000 }
gfCNCPoint1[12422] = {X 280.8083, Y 46.8619, Z -1.3333, A 0.000, B 0.000, C 0.000 }
gfCNCPoint1[12423] = {X 280.4907, Y 45.9723, Z -1.3333, A 0.000, B 0.000, C 0.000 }
gfCNCPoint1[12424] = {X 280.3778, Y 45.0345, Z -1.3333, A 0.000, B 0.000, C 0.000 }
gfCNCPoint1[12425] = {X 280.3777, Y 44.2074, Z -1.3333, A 0.000, B 0.000, C 0.000 }
gfCNCPoint1[12426] = {X 280.4833, Y 43.2867, Z -1.3333, A 0.000, B 0.000, C 0.000 }
gfCNCPoint1[12427] = {X 280.7841, Y 42.4100, Z -1.3333, A 0.000, B 0.000, C 0.000 }
gfCNCPoint1[12428] = {X 281.2660, Y 41.6184, Z -1.3333, A 0.000, B 0.000, C 0.000 }
gfCNCPoint1[12429] = {X 281.9065, Y 40.9485, Z -1.3333, A 0.000, B 0.000, C 0.000 }
gfCNCPoint1[12430] = {X 281.9063, Y 28.5932, Z -1.3333, A 0.000, B 0.000, C 0.000 }
gfCNCPoint1[12431] = {X 277.9063, Y 28.5933, Z -1.3333, A 0.000, B 0.000, C 0.000 }
gfCNCPoint1[12432] = {X 281.9863, Y 28.5932, Z -1.3333, A 0.000, B 0.000, C 0.000 }
gfCNCPoint1[12433] = {X 281.9861, Y 16.1999, Z -1.3333, A 0.000, B 0.000, C 0.000 }
gfCNCPoint1[12434] = {X 281.3481, Y 15.5501, Z -1.3333, A 0.000, B 0.000, C 0.000 }
gfCNCPoint1[12435] = {X 280.8668, Y 14.7771, Z -1.3333, A 0.000, B 0.000, C 0.000 }
gfCNCPoint1[12436] = {X 280.5652, Y 13.9179, Z -1.3333, A 0.000, B 0.000, C 0.000 }
gfCNCPoint1[12437] = {X 280.4578, Y 13.0136, Z -1.3333, A 0.000, B 0.000, C 0.000 }
gfCNCPoint1[12438] = {X 280.4577, Y 12.1868, Z -1.3333, A 0.000, B 0.000, C 0.000 }
gfCNCPoint1[12439] = {X 280.5620, Y 11.2611, Z -1.3333, A 0.000, B 0.000, C 0.000 }
gfCNCPoint1[12440] = {X 280.8696, Y 10.3819, Z -1.3333, A 0.000, B 0.000, C 0.000 }
gfCNCPoint1[12441] = {X 281.3652, Y 9.5931, Z -1.3333, A 0.000, B 0.000, C 0.000 }
gfCNCPoint1[12442] = {X 282.0240, Y 8.9344, Z -1.3333, A 0.000, B 0.000, C 0.000 }
gfCNCPoint1[12443] = {X 282.8127, Y 8.4388, Z -1.3333, A 0.000, B 0.000, C 0.000 }
gfCNCPoint1[12444] = {X 283.6920, Y 8.1311, Z -1.3333, A 0.000, B 0.000, C 0.000 }
gfCNCPoint1[12445] = {X 284.6177, Y 8.0268, Z -1.3333, A 0.000, B 0.000, C 0.000 }
gfCNCPoint1[12446] = {X 291.0611, Y 8.0268, Z -1.3333, A 0.000, B 0.000, C 0.000 }
gfCNCPoint1[12447] = {X 291.9868, Y 8.1311, Z -1.3333, A 0.000, B 0.000, C 0.000 }
gfCNCPoint1[12448] = {X 292.8661, Y 8.4388, Z -1.3333, A 0.000, B 0.000, C 0.000 }
gfCNCPoint1[12449] = {X 293.6549, Y 8.9344, Z -1.3333, A 0.000, B 0.000, C 0.000 }
gfCNCPoint1[12450] = {X 294.3136, Y 9.5931, Z -1.3333, A 0.000, B 0.000, C 0.000 }
gfCNCPoint1[12451] = {X 294.8092, Y 10.3819, Z -1.3333, A 0.000, B 0.000, C 0.000 }
gfCNCPoint1[12452] = {X 295.1168, Y 11.2611, Z -1.3333, A 0.000, B 0.000, C 0.000 }
gfCNCPoint1[12453] = {X 295.2211, Y 12.1868, Z -1.3333, A 0.000, B 0.000, C 0.000 }
gfCNCPoint1[12454] = {X 295.2211, Y 12.9781, Z -1.3333, A 0.000, B 0.000, C 0.000 }
gfCNCPoint1[12455] = {X 295.1254, Y 13.8655, Z -1.3333, A 0.000, B 0.000, C 0.000 }
gfCNCPoint1[12456] = {X 294.8426, Y 14.7120, Z -1.3333, A 0.000, B 0.000, C 0.000 }
gfCNCPoint1[12457] = {X 294.3857, Y 15.4786, Z -1.3333, A 0.000, B 0.000, C 0.000 }
gfCNCPoint1[12458] = {X 293.7758, Y 16.1302, Z -1.3333, A 0.000, B 0.000, C 0.000 }
gfCNCPoint1[12459] = {X 293.6924, Y 16.2002, Z -1.3333, A 0.000, B 0.000, C 0.000 }
gfCNCPoint1[12460] = {X 293.6938, Y 22.3568, Z -1.3333, A 0.000, B 0.000, C 0.000 }
gfCNCPoint1[12461] = {X 302.9200, Y 22.3565, Z -1.3333, A 0.000, B 0.000, C 0.000 }
gfCNCPoint1[12462] = {X 302.9249, Y 16.2033, Z -1.3333, A 0.000, B 0.000, C 0.000 }
gfCNCPoint1[12463] = {X 302.2855, Y 15.5536, Z -1.3333, A 0.000, B 0.000, C 0.000 }
gfCNCPoint1[12464] = {X 301.8029, Y 14.7802, Z -1.3333, A 0.000, B 0.000, C 0.000 }
gfCNCPoint1[12465] = {X 301.5004, Y 13.9203, Z -1.3333, A 0.000, B 0.000, C 0.000 }
gfCNCPoint1[12466] = {X 301.3924, Y 13.0151, Z -1.3333, A 0.000, B 0.000, C 0.000 }
gfCNCPoint1[12467] = {X 301.3923, Y 12.1868, Z -1.3333, A 0.000, B 0.000, C 0.000 }
gfCNCPoint1[12468] = {X 301.4966, Y 11.2611, Z -1.3333, A 0.000, B 0.000, C 0.000 }
gfCNCPoint1[12469] = {X 301.8042, Y 10.3819, Z -1.3333, A 0.000, B 0.000, C 0.000 }
gfCNCPoint1[12470] = {X 302.2998, Y 9.5931, Z -1.3333, A 0.000, B 0.000, C 0.000 }
gfCNCPoint1[12471] = {X 302.9585, Y 8.9344, Z -1.3333, A 0.000, B 0.000, C 0.000 }
gfCNCPoint1[12472] = {X 303.7473, Y 8.4388, Z -1.3333, A 0.000, B 0.000, C 0.000 }
gfCNCPoint1[12473] = {X 304.6266, Y 8.1311, Z -1.3333, A 0.000, B 0.000, C 0.000 }
gfCNCPoint1[12474] = {X 305.5523, Y 8.0268, Z -1.3333, A 0.000, B 0.000, C 0.000 }
gfCNCPoint1[12475] = {X 311.9957, Y 8.0268, Z -1.3333, A 0.000, B 0.000, C 0.000 }
gfCNCPoint1[12476] = {X 312.9214, Y 8.1311, Z -1.3333, A 0.000, B 0.000, C 0.000 }
gfCNCPoint1[12477] = {X 313.8007, Y 8.4388, Z -1.3333, A 0.000, B 0.000, C 0.000 }
gfCNCPoint1[12478] = {X 314.5894, Y 8.9344, Z -1.3333, A 0.000, B 0.000, C 0.000 }
gfCNCPoint1[12479] = {X 315.2481, Y 9.5931, Z -1.3333, A 0.000, B 0.000, C 0.000 }
gfCNCPoint1[12480] = {X 315.7438, Y 10.3819, Z -1.3333, A 0.000, B 0.000, C 0.000 }
gfCNCPoint1[12481] = {X 316.0514, Y 11.2611, Z -1.3333, A 0.000, B 0.000, C 0.000 }
gfCNCPoint1[12482] = {X 316.1557, Y 12.1868, Z -1.3333, A 0.000, B 0.000, C 0.000 }
gfCNCPoint1[12483] = {X 316.1557, Y 12.9781, Z -1.3333, A 0.000, B 0.000, C 0.000 }
gfCNCPoint1[12484] = {X 316.0541, Y 13.8917, Z -1.3333, A 0.000, B 0.000, C 0.000 }
gfCNCPoint1[12485] = {X 315.7544, Y 14.7608, Z -1.3333, A 0.000, B 0.000, C 0.000 }
gfCNCPoint1[12486] = {X 315.2711, Y 15.5427, Z -1.3333, A 0.000, B 0.000, C 0.000 }
gfCNCPoint1[12487] = {X 314.6279, Y 16.1994, Z -1.3333, A 0.000, B 0.000, C 0.000 }
gfCNCPoint1[12488] = {X 314.6269, Y 40.9892, Z -1.3333, A 0.000, B 0.000, C 0.000 }
gfCNCPoint1[12489] = {X 314.6830, Y 41.0332, Z -1.3333, A 0.000, B 0.000, C 0.000 }
gfCNCPoint1[12490] = {X 315.2985, Y 41.6795, Z -1.3333, A 0.000, B 0.000, C 0.000 }
gfCNCPoint1[12491] = {X 315.7620, Y 42.4422, Z -1.3333, A 0.000, B 0.000, C 0.000 }
gfCNCPoint1[12492] = {X 316.0521, Y 43.2862, Z -1.3333, A 0.000, B 0.000, C 0.000 }
gfCNCPoint1[12493] = {X 316.1556, Y 44.1727, Z -1.3333, A 0.000, B 0.000, C 0.000 }
gfCNCPoint1[12494] = {X 316.1557, Y 45.0000, Z -1.3333, A 0.000, B 0.000, C 0.000 }
gfCNCPoint1[12495] = {X 316.0514, Y 45.9257, Z -1.3333, A 0.000, B 0.000, C 0.000 }
gfCNCPoint1[12496] = {X 315.7438, Y 46.8050, Z -1.3333, A 0.000, B 0.000, C 0.000 }
gfCNCPoint1[12497] = {X 315.2481, Y 47.5937, Z -1.3333, A 0.000, B 0.000, C 0.000 }
gfCNCPoint1[12498] = {X 314.5894, Y 48.2524, Z -1.3333, A 0.000, B 0.000, C 0.000 }
gfCNCPoint1[12499] = {X 313.8007, Y 48.7480, Z -1.3333, A 0.000, B 0.000, C 0.000 }
gfCNCPoint1[12500] = {X 312.9214, Y 49.0557, Z -1.3333, A 0.000, B 0.000, C 0.000 }
gfCNCPoint1[12501] = {X 311.9957, Y 49.1600, Z -1.3333, A 0.000, B 0.000, C 0.000 }
gfCNCPoint1[12502] = {X 305.5523, Y 49.1600, Z -1.3333, A 0.000, B 0.000, C 0.000 }
gfCNCPoint1[12503] = {X 304.6312, Y 49.0568, Z -1.3333, A 0.000, B 0.000, C 0.000 }
gfCNCPoint1[12504] = {X 303.7559, Y 48.7522, Z -1.3333, A 0.000, B 0.000, C 0.000 }
gfCNCPoint1[12505] = {X 302.9698, Y 48.2613, Z -1.3333, A 0.000, B 0.000, C 0.000 }
gfCNCPoint1[12506] = {X 302.3118, Y 47.6087, Z -1.3333, A 0.000, B 0.000, C 0.000 }
gfCNCPoint1[12507] = {X 301.8147, Y 46.8265, Z -1.3333, A 0.000, B 0.000, C 0.000 }
gfCNCPoint1[12508] = {X 301.5030, Y 45.9537, Z -1.3333, A 0.000, B 0.000, C 0.000 }
gfCNCPoint1[12509] = {X 301.3924, Y 45.0335, Z -1.3333, A 0.000, B 0.000, C 0.000 }
gfCNCPoint1[12510] = {X 301.3923, Y 44.2050, Z -1.3333, A 0.000, B 0.000, C 0.000 }
gfCNCPoint1[12511] = {X 301.5105, Y 43.2838, Z -1.3333, A 0.000, B 0.000, C 0.000 }
gfCNCPoint1[12512] = {X 301.8144, Y 42.4063, Z -1.3333, A 0.000, B 0.000, C 0.000 }
gfCNCPoint1[12513] = {X 302.2914, Y 41.6094, Z -1.3333, A 0.000, B 0.000, C 0.000 }
gfCNCPoint1[12514] = {X 302.9211, Y 40.9269, Z -1.3333, A 0.000, B 0.000, C 0.000 }
gfCNCPoint1[12515] = {X 302.9211, Y 33.8743, Z -1.3333, A 0.000, B 0.000, C 0.000 }
gfCNCPoint1[12516] = {X 293.6935, Y 33.8743, Z -1.3333, A 0.000, B 0.000, C 0.000 }
gfCNCPoint1[12517] = {X 293.6924, Y 40.9769, Z -1.3333, A 0.000, B 0.000, C 0.000 }
gfCNCPoint1[12518] = {X 294.3307, Y 41.6399, Z -1.3333, A 0.000, B 0.000, C 0.000 }
gfCNCPoint1[12519] = {X 294.8117, Y 42.4244, Z -1.3333, A 0.000, B 0.000, C 0.000 }
gfCNCPoint1[12520] = {X 295.1132, Y 43.2939, Z -1.3333, A 0.000, B 0.000, C 0.000 }
gfCNCPoint1[12521] = {X 295.2211, Y 44.2078, Z -1.3333, A 0.000, B 0.000, C 0.000 }
gfCNCPoint1[12522] = {X 295.2211, Y 45.0000, Z -1.3333, A 0.000, B 0.000, C 0.000 }
gfCNCPoint1[12523] = {X 295.1168, Y 45.9257, Z -1.3333, A 0.000, B 0.000, C 0.000 }
gfCNCPoint1[12524] = {X 294.8092, Y 46.8050, Z -1.3333, A 0.000, B 0.000, C 0.000 }
gfCNCPoint1[12525] = {X 294.3136, Y 47.5937, Z -1.3333, A 0.000, B 0.000, C 0.000 }
gfCNCPoint1[12526] = {X 293.6549, Y 48.2524, Z -1.3333, A 0.000, B 0.000, C 0.000 }
gfCNCPoint1[12527] = {X 292.8661, Y 48.7480, Z -1.3333, A 0.000, B 0.000, C 0.000 }
gfCNCPoint1[12528] = {X 291.9868, Y 49.0557, Z -1.3333, A 0.000, B 0.000, C 0.000 }
gfCNCPoint1[12529] = {X 291.0611, Y 49.1600, Z -1.3333, A 0.000, B 0.000, C 0.000 }
gfCNCPoint1[12530] = {X 284.6177, Y 49.1600, Z -1.3333, A 0.000, B 0.000, C 0.000 }
gfCNCPoint1[12531] = {X 283.6967, Y 49.0568, Z -1.3333, A 0.000, B 0.000, C 0.000 }
gfCNCPoint1[12532] = {X 282.8214, Y 48.7522, Z -1.3333, A 0.000, B 0.000, C 0.000 }
gfCNCPoint1[12533] = {X 282.0353, Y 48.2615, Z -1.3333, A 0.000, B 0.000, C 0.000 }
gfCNCPoint1[12534] = {X 281.3774, Y 47.6088, Z -1.3333, A 0.000, B 0.000, C 0.000 }
gfCNCPoint1[12535] = {X 280.8802, Y 46.8267, Z -1.3333, A 0.000, B 0.000, C 0.000 }
gfCNCPoint1[12536] = {X 280.5685, Y 45.9540, Z -1.3333, A 0.000, B 0.000, C 0.000 }
gfCNCPoint1[12537] = {X 280.4578, Y 45.0339, Z -1.3333, A 0.000, B 0.000, C 0.000 }
gfCNCPoint1[12538] = {X 280.4577, Y 44.2079, Z -1.3333, A 0.000, B 0.000, C 0.000 }
gfCNCPoint1[12539] = {X 280.5634, Y 43.2953, Z -1.3333, A 0.000, B 0.000, C 0.000 }
gfCNCPoint1[12540] = {X 280.8645, Y 42.4272, Z -1.3333, A 0.000, B 0.000, C 0.000 }
gfCNCPoint1[12541] = {X 281.3465, Y 41.6451, Z -1.3333, A 0.000, B 0.000, C 0.000 }
gfCNCPoint1[12542] = {X 281.9865, Y 40.9860, Z -1.3333, A 0.000, B 0.000, C 0.000 }
gfCNCPoint1[12543] = {X 281.9863, Y 28.5932, Z -1.3333, A 0.000, B 0.000, C 0.000 }
gfCNCPoint1[12544] = {X 277.9863, Y 28.5933, Z -1.3333, A 0.000, B 0.000, C 0.000 }
gfCNCPoint1[12545] = {X 282.0663, Y 28.5932, Z -1.3333, A 0.000, B 0.000, C 0.000 }
gfCNCPoint1[12546] = {X 282.0661, Y 16.1617, Z -1.3333, A 0.000, B 0.000, C 0.000 }
gfCNCPoint1[12547] = {X 281.4286, Y 15.5229, Z -1.3333, A 0.000, B 0.000, C 0.000 }
gfCNCPoint1[12548] = {X 280.9472, Y 14.7595, Z -1.3333, A 0.000, B 0.000, C 0.000 }
gfCNCPoint1[12549] = {X 280.6453, Y 13.9090, Z -1.3333, A 0.000, B 0.000, C 0.000 }
gfCNCPoint1[12550] = {X 280.5378, Y 13.0129, Z -1.3333, A 0.000, B 0.000, C 0.000 }
gfCNCPoint1[12551] = {X 280.5377, Y 12.1868, Z -1.3333, A 0.000, B 0.000, C 0.000 }
gfCNCPoint1[12552] = {X 280.6400, Y 11.2789, Z -1.3333, A 0.000, B 0.000, C 0.000 }
gfCNCPoint1[12553] = {X 280.9417, Y 10.4166, Z -1.3333, A 0.000, B 0.000, C 0.000 }
gfCNCPoint1[12554] = {X 281.4278, Y 9.6430, Z -1.3333, A 0.000, B 0.000, C 0.000 }
gfCNCPoint1[12555] = {X 282.0738, Y 8.9969, Z -1.3333, A 0.000, B 0.000, C 0.000 }
gfCNCPoint1[12556] = {X 282.8474, Y 8.5109, Z -1.3333, A 0.000, B 0.000, C 0.000 }
gfCNCPoint1[12557] = {X 283.7098, Y 8.2091, Z -1.3333, A 0.000, B 0.000, C 0.000 }
gfCNCPoint1[12558] = {X 284.6177, Y 8.1068, Z -1.3333, A 0.000, B 0.000, C 0.000 }
gfCNCPoint1[12559] = {X 291.0611, Y 8.1068, Z -1.3333, A 0.000, B 0.000, C 0.000 }
gfCNCPoint1[12560] = {X 291.9690, Y 8.2091, Z -1.3333, A 0.000, B 0.000, C 0.000 }
gfCNCPoint1[12561] = {X 292.8314, Y 8.5109, Z -1.3333, A 0.000, B 0.000, C 0.000 }
gfCNCPoint1[12562] = {X 293.6050, Y 8.9969, Z -1.3333, A 0.000, B 0.000, C 0.000 }
gfCNCPoint1[12563] = {X 294.2510, Y 9.6430, Z -1.3333, A 0.000, B 0.000, C 0.000 }
gfCNCPoint1[12564] = {X 294.7371, Y 10.4166, Z -1.3333, A 0.000, B 0.000, C 0.000 }
gfCNCPoint1[12565] = {X 295.0388, Y 11.2789, Z -1.3333, A 0.000, B 0.000, C 0.000 }
gfCNCPoint1[12566] = {X 295.1411, Y 12.1868, Z -1.3333, A 0.000, B 0.000, C 0.000 }
gfCNCPoint1[12567] = {X 295.1411, Y 12.9781, Z -1.3333, A 0.000, B 0.000, C 0.000 }
gfCNCPoint1[12568] = {X 295.0472, Y 13.8484, Z -1.3333, A 0.000, B 0.000, C 0.000 }
gfCNCPoint1[12569] = {X 294.7698, Y 14.6786, Z -1.3333, A 0.000, B 0.000, C 0.000 }
gfCNCPoint1[12570] = {X 294.3217, Y 15.4305, Z -1.3333, A 0.000, B 0.000, C 0.000 }
gfCNCPoint1[12571] = {X 293.7236, Y 16.0696, Z -1.3333, A 0.000, B 0.000, C 0.000 }
gfCNCPoint1[12572] = {X 293.6663, Y 16.1180, Z -1.3333, A 0.000, B 0.000, C 0.000 }
gfCNCPoint1[12573] = {X 293.6082, Y 16.1653, Z -1.3333, A 0.000, B 0.000, C 0.000 }
gfCNCPoint1[12574] = {X 293.6124, Y 16.2002, Z -1.3333, A 0.000, B 0.000, C 0.000 }
gfCNCPoint1[12575] = {X 293.6138, Y 22.4372, Z -1.3333, A 0.000, B 0.000, C 0.000 }
gfCNCPoint1[12576] = {X 293.7675, Y 22.4365, Z -1.3333, A 0.000, B 0.000, C 0.000 }
gfCNCPoint1[12577] = {X 302.9999, Y 22.4365, Z -1.3333, A 0.000, B 0.000, C 0.000 }
gfCNCPoint1[12578] = {X 303.0049, Y 16.1651, Z -1.3333, A 0.000, B 0.000, C 0.000 }
gfCNCPoint1[12579] = {X 302.9467, Y 16.1177, Z -1.3333, A 0.000, B 0.000, C 0.000 }
gfCNCPoint1[12580] = {X 302.8894, Y 16.0693, Z -1.3333, A 0.000, B 0.000, C 0.000 }
gfCNCPoint1[12581] = {X 302.2969, Y 15.4375, Z -1.3333, A 0.000, B 0.000, C 0.000 }
gfCNCPoint1[12582] = {X 301.8511, Y 14.6949, Z -1.3333, A 0.000, B 0.000, C 0.000 }
gfCNCPoint1[12583] = {X 301.5720, Y 13.8748, Z -1.3333, A 0.000, B 0.000, C 0.000 }
gfCNCPoint1[12584] = {X 301.4724, Y 13.0144, Z -1.3333, A 0.000, B 0.000, C 0.000 }
gfCNCPoint1[12585] = {X 301.4723, Y 12.1868, Z -1.3333, A 0.000, B 0.000, C 0.000 }
gfCNCPoint1[12586] = {X 301.5745, Y 11.2789, Z -1.3333, A 0.000, B 0.000, C 0.000 }
gfCNCPoint1[12587] = {X 301.8763, Y 10.4166, Z -1.3333, A 0.000, B 0.000, C 0.000 }
gfCNCPoint1[12588] = {X 302.3624, Y 9.6430, Z -1.3333, A 0.000, B 0.000, C 0.000 }
gfCNCPoint1[12589] = {X 303.0084, Y 8.9969, Z -1.3333, A 0.000, B 0.000, C 0.000 }
gfCNCPoint1[12590] = {X 303.7820, Y 8.5109, Z -1.3333, A 0.000, B 0.000, C 0.000 }
gfCNCPoint1[12591] = {X 304.6444, Y 8.2091, Z -1.3333, A 0.000, B 0.000, C 0.000 }
gfCNCPoint1[12592] = {X 305.5523, Y 8.1068, Z -1.3333, A 0.000, B 0.000, C 0.000 }
gfCNCPoint1[12593] = {X 311.9957, Y 8.1068, Z -1.3333, A 0.000, B 0.000, C 0.000 }
gfCNCPoint1[12594] = {X 312.9036, Y 8.2091, Z -1.3333, A 0.000, B 0.000, C 0.000 }
gfCNCPoint1[12595] = {X 313.7660, Y 8.5109, Z -1.3333, A 0.000, B 0.000, C 0.000 }
gfCNCPoint1[12596] = {X 314.5396, Y 8.9969, Z -1.3333, A 0.000, B 0.000, C 0.000 }
gfCNCPoint1[12597] = {X 315.1856, Y 9.6430, Z -1.3333, A 0.000, B 0.000, C 0.000 }
gfCNCPoint1[12598] = {X 315.6717, Y 10.4166, Z -1.3333, A 0.000, B 0.000, C 0.000 }
gfCNCPoint1[12599] = {X 315.9734, Y 11.2789, Z -1.3333, A 0.000, B 0.000, C 0.000 }
gfCNCPoint1[12600] = {X 316.0757, Y 12.1868, Z -1.3333, A 0.000, B 0.000, C 0.000 }
gfCNCPoint1[12601] = {X 316.0757, Y 12.9781, Z -1.3333, A 0.000, B 0.000, C 0.000 }
gfCNCPoint1[12602] = {X 315.9818, Y 13.8483, Z -1.3333, A 0.000, B 0.000, C 0.000 }
gfCNCPoint1[12603] = {X 315.7045, Y 14.6785, Z -1.3333, A 0.000, B 0.000, C 0.000 }
gfCNCPoint1[12604] = {X 315.2564, Y 15.4304, Z -1.3333, A 0.000, B 0.000, C 0.000 }
gfCNCPoint1[12605] = {X 314.6583, Y 16.0695, Z -1.3333, A 0.000, B 0.000, C 0.000 }
gfCNCPoint1[12606] = {X 314.6039, Y 16.1155, Z -1.3333, A 0.000, B 0.000, C 0.000 }
gfCNCPoint1[12607] = {X 314.5487, Y 16.1606, Z -1.3333, A 0.000, B 0.000, C 0.000 }
gfCNCPoint1[12608] = {X 314.5469, Y 41.0281, Z -1.3333, A 0.000, B 0.000, C 0.000 }
gfCNCPoint1[12609] = {X 314.6336, Y 41.0962, Z -1.3333, A 0.000, B 0.000, C 0.000 }
gfCNCPoint1[12610] = {X 315.2363, Y 41.7299, Z -1.3333, A 0.000, B 0.000, C 0.000 }
gfCNCPoint1[12611] = {X 315.6902, Y 42.4775, Z -1.3333, A 0.000, B 0.000, C 0.000 }
gfCNCPoint1[12612] = {X 315.9743, Y 43.3047, Z -1.3333, A 0.000, B 0.000, C 0.000 }
gfCNCPoint1[12613] = {X 316.0756, Y 44.1734, Z -1.3333, A 0.000, B 0.000, C 0.000 }
gfCNCPoint1[12614] = {X 316.0757, Y 45.0000, Z -1.3333, A 0.000, B 0.000, C 0.000 }
gfCNCPoint1[12615] = {X 315.9734, Y 45.9079, Z -1.3333, A 0.000, B 0.000, C 0.000 }
gfCNCPoint1[12616] = {X 315.6717, Y 46.7702, Z -1.3333, A 0.000, B 0.000, C 0.000 }
gfCNCPoint1[12617] = {X 315.1856, Y 47.5438, Z -1.3333, A 0.000, B 0.000, C 0.000 }
gfCNCPoint1[12618] = {X 314.5396, Y 48.1899, Z -1.3333, A 0.000, B 0.000, C 0.000 }
gfCNCPoint1[12619] = {X 313.7660, Y 48.6760, Z -1.3333, A 0.000, B 0.000, C 0.000 }
gfCNCPoint1[12620] = {X 312.9036, Y 48.9777, Z -1.3333, A 0.000, B 0.000, C 0.000 }
gfCNCPoint1[12621] = {X 311.9957, Y 49.0800, Z -1.3333, A 0.000, B 0.000, C 0.000 }
gfCNCPoint1[12622] = {X 305.5523, Y 49.0800, Z -1.3333, A 0.000, B 0.000, C 0.000 }
gfCNCPoint1[12623] = {X 304.6489, Y 48.9787, Z -1.3333, A 0.000, B 0.000, C 0.000 }
gfCNCPoint1[12624] = {X 303.7905, Y 48.6800, Z -1.3333, A 0.000, B 0.000, C 0.000 }
gfCNCPoint1[12625] = {X 303.0194, Y 48.1986, Z -1.3333, A 0.000, B 0.000, C 0.000 }
gfCNCPoint1[12626] = {X 302.3741, Y 47.5585, Z -1.3333, A 0.000, B 0.000, C 0.000 }
gfCNCPoint1[12627] = {X 301.8865, Y 46.7914, Z -1.3333, A 0.000, B 0.000, C 0.000 }
gfCNCPoint1[12628] = {X 301.5809, Y 45.9353, Z -1.3333, A 0.000, B 0.000, C 0.000 }
gfCNCPoint1[12629] = {X 301.4724, Y 45.0328, Z -1.3333, A 0.000, B 0.000, C 0.000 }
gfCNCPoint1[12630] = {X 301.4723, Y 44.2069, Z -1.3333, A 0.000, B 0.000, C 0.000 }
gfCNCPoint1[12631] = {X 301.5904, Y 43.2934, Z -1.3333, A 0.000, B 0.000, C 0.000 }
gfCNCPoint1[12632] = {X 301.8946, Y 42.4238, Z -1.3333, A 0.000, B 0.000, C 0.000 }
gfCNCPoint1[12633] = {X 302.3716, Y 41.6358, Z -1.3333, A 0.000, B 0.000, C 0.000 }
gfCNCPoint1[12634] = {X 303.0011, Y 40.9632, Z -1.3333, A 0.000, B 0.000, C 0.000 }
gfCNCPoint1[12635] = {X 303.0011, Y 33.7943, Z -1.3333, A 0.000, B 0.000, C 0.000 }
gfCNCPoint1[12636] = {X 293.6135, Y 33.7943, Z -1.3333, A 0.000, B 0.000, C 0.000 }
gfCNCPoint1[12637] = {X 293.6124, Y 41.0145, Z -1.3333, A 0.000, B 0.000, C 0.000 }
gfCNCPoint1[12638] = {X 294.2502, Y 41.6668, Z -1.3333, A 0.000, B 0.000, C 0.000 }
gfCNCPoint1[12639] = {X 294.7314, Y 42.4418, Z -1.3333, A 0.000, B 0.000, C 0.000 }
gfCNCPoint1[12640] = {X 295.0332, Y 43.3027, Z -1.3333, A 0.000, B 0.000, C 0.000 }
gfCNCPoint1[12641] = {X 295.1411, Y 44.2085, Z -1.3333, A 0.000, B 0.000, C 0.000 }
gfCNCPoint1[12642] = {X 295.1411, Y 45.0000, Z -1.3333, A 0.000, B 0.000, C 0.000 }
gfCNCPoint1[12643] = {X 295.0388, Y 45.9079, Z -1.3333, A 0.000, B 0.000, C 0.000 }
gfCNCPoint1[12644] = {X 294.7371, Y 46.7702, Z -1.3333, A 0.000, B 0.000, C 0.000 }
gfCNCPoint1[12645] = {X 294.2510, Y 47.5438, Z -1.3333, A 0.000, B 0.000, C 0.000 }
gfCNCPoint1[12646] = {X 293.6050, Y 48.1899, Z -1.3333, A 0.000, B 0.000, C 0.000 }
gfCNCPoint1[12647] = {X 292.8314, Y 48.6760, Z -1.3333, A 0.000, B 0.000, C 0.000 }
gfCNCPoint1[12648] = {X 291.9690, Y 48.9777, Z -1.3333, A 0.000, B 0.000, C 0.000 }
gfCNCPoint1[12649] = {X 291.0611, Y 49.0800, Z -1.3333, A 0.000, B 0.000, C 0.000 }
gfCNCPoint1[12650] = {X 284.6177, Y 49.0800, Z -1.3333, A 0.000, B 0.000, C 0.000 }
gfCNCPoint1[12651] = {X 283.7144, Y 48.9788, Z -1.3333, A 0.000, B 0.000, C 0.000 }
gfCNCPoint1[12652] = {X 282.8560, Y 48.6801, Z -1.3333, A 0.000, B 0.000, C 0.000 }
gfCNCPoint1[12653] = {X 282.0850, Y 48.1987, Z -1.3333, A 0.000, B 0.000, C 0.000 }
gfCNCPoint1[12654] = {X 281.4397, Y 47.5587, Z -1.3333, A 0.000, B 0.000, C 0.000 }
gfCNCPoint1[12655] = {X 280.9521, Y 46.7916, Z -1.3333, A 0.000, B 0.000, C 0.000 }
gfCNCPoint1[12656] = {X 280.6464, Y 45.9356, Z -1.3333, A 0.000, B 0.000, C 0.000 }
gfCNCPoint1[12657] = {X 280.5378, Y 45.0332, Z -1.3333, A 0.000, B 0.000, C 0.000 }
gfCNCPoint1[12658] = {X 280.5377, Y 44.2084, Z -1.3333, A 0.000, B 0.000, C 0.000 }
gfCNCPoint1[12659] = {X 280.6435, Y 43.3040, Z -1.3333, A 0.000, B 0.000, C 0.000 }
gfCNCPoint1[12660] = {X 280.9448, Y 42.4446, Z -1.3333, A 0.000, B 0.000, C 0.000 }
gfCNCPoint1[12661] = {X 281.4270, Y 41.6721, Z -1.3333, A 0.000, B 0.000, C 0.000 }
gfCNCPoint1[12662] = {X 282.0665, Y 41.0238, Z -1.3333, A 0.000, B 0.000, C 0.000 }
gfCNCPoint1[12663] = {X 282.0663, Y 28.5932, Z -1.3333, A 0.000, B 0.000, C 0.000 }
gfCNCPoint1[12664] = {X 278.0663, Y 28.5933, Z -1.3333, A 0.000, B 0.000, C 0.000 }
gfCNCPoint1[12665] = {X 282.1463, Y 28.5932, Z -1.3333, A 0.000, B 0.000, C 0.000 }
gfCNCPoint1[12666] = {X 282.1461, Y 16.1231, Z -1.3333, A 0.000, B 0.000, C 0.000 }
gfCNCPoint1[12667] = {X 281.5037, Y 15.4887, Z -1.3333, A 0.000, B 0.000, C 0.000 }
gfCNCPoint1[12668] = {X 281.0200, Y 14.7264, Z -1.3333, A 0.000, B 0.000, C 0.000 }
gfCNCPoint1[12669] = {X 280.7195, Y 13.8750, Z -1.3333, A 0.000, B 0.000, C 0.000 }
gfCNCPoint1[12670] = {X 280.6177, Y 12.9779, Z -1.3333, A 0.000, B 0.000, C 0.000 }
gfCNCPoint1[12671] = {X 280.6177, Y 12.1868, Z -1.3333, A 0.000, B 0.000, C 0.000 }
gfCNCPoint1[12672] = {X 280.7180, Y 11.2967, Z -1.3333, A 0.000, B 0.000, C 0.000 }
gfCNCPoint1[12673] = {X 281.0138, Y 10.4513, Z -1.3333, A 0.000, B 0.000, C 0.000 }
gfCNCPoint1[12674] = {X 281.4903, Y 9.6929, Z -1.3333, A 0.000, B 0.000, C 0.000 }
gfCNCPoint1[12675] = {X 282.1237, Y 9.0595, Z -1.3333, A 0.000, B 0.000, C 0.000 }
gfCNCPoint1[12676] = {X 282.8821, Y 8.5829, Z -1.3333, A 0.000, B 0.000, C 0.000 }
gfCNCPoint1[12677] = {X 283.7276, Y 8.2871, Z -1.3333, A 0.000, B 0.000, C 0.000 }
gfCNCPoint1[12678] = {X 284.6177, Y 8.1868, Z -1.3333, A 0.000, B 0.000, C 0.000 }
gfCNCPoint1[12679] = {X 291.0611, Y 8.1868, Z -1.3333, A 0.000, B 0.000, C 0.000 }
gfCNCPoint1[12680] = {X 291.9512, Y 8.2871, Z -1.3333, A 0.000, B 0.000, C 0.000 }
gfCNCPoint1[12681] = {X 292.7967, Y 8.5829, Z -1.3333, A 0.000, B 0.000, C 0.000 }
gfCNCPoint1[12682] = {X 293.5551, Y 9.0595, Z -1.3333, A 0.000, B 0.000, C 0.000 }
gfCNCPoint1[12683] = {X 294.1885, Y 9.6929, Z -1.3333, A 0.000, B 0.000, C 0.000 }
gfCNCPoint1[12684] = {X 294.6650, Y 10.4513, Z -1.3333, A 0.000, B 0.000, C 0.000 }
gfCNCPoint1[12685] = {X 294.9608, Y 11.2967, Z -1.3333, A 0.000, B 0.000, C 0.000 }
gfCNCPoint1[12686] = {X 295.0611, Y 12.1868, Z -1.3333, A 0.000, B 0.000, C 0.000 }
gfCNCPoint1[12687] = {X 295.0609, Y 13.0192, Z -1.3333, A 0.000, B 0.000, C 0.000 }
gfCNCPoint1[12688] = {X 294.9624, Y 13.8614, Z -1.3333, A 0.000, B 0.000, C 0.000 }
gfCNCPoint1[12689] = {X 294.6885, Y 14.6639, Z -1.3333, A 0.000, B 0.000, C 0.000 }
gfCNCPoint1[12690] = {X 294.2516, Y 15.3907, Z -1.3333, A 0.000, B 0.000, C 0.000 }
gfCNCPoint1[12691] = {X 293.6714, Y 16.0090, Z -1.3333, A 0.000, B 0.000, C 0.000 }
gfCNCPoint1[12692] = {X 293.5953, Y 16.0729, Z -1.3333, A 0.000, B 0.000, C 0.000 }
gfCNCPoint1[12693] = {X 293.5177, Y 16.1348, Z -1.3333, A 0.000, B 0.000, C 0.000 }
gfCNCPoint1[12694] = {X 293.5324, Y 16.1918, Z -1.3333, A 0.000, B 0.000, C 0.000 }
gfCNCPoint1[12695] = {X 293.5338, Y 22.5176, Z -1.3333, A 0.000, B 0.000, C 0.000 }
gfCNCPoint1[12696] = {X 293.7676, Y 22.5165, Z -1.3333, A 0.000, B 0.000, C 0.000 }
gfCNCPoint1[12697] = {X 303.0799, Y 22.5180, Z -1.3333, A 0.000, B 0.000, C 0.000 }
gfCNCPoint1[12698] = {X 303.0806, Y 16.1919, Z -1.3333, A 0.000, B 0.000, C 0.000 }
gfCNCPoint1[12699] = {X 303.0955, Y 16.1346, Z -1.3333, A 0.000, B 0.000, C 0.000 }
gfCNCPoint1[12700] = {X 303.0178, Y 16.0726, Z -1.3333, A 0.000, B 0.000, C 0.000 }
gfCNCPoint1[12701] = {X 302.9417, Y 16.0087, Z -1.3333, A 0.000, B 0.000, C 0.000 }
gfCNCPoint1[12702] = {X 302.3553, Y 15.3821, Z -1.3333, A 0.000, B 0.000, C 0.000 }
gfCNCPoint1[12703] = {X 301.9161, Y 14.6449, Z -1.3333, A 0.000, B 0.000, C 0.000 }
gfCNCPoint1[12704] = {X 301.6443, Y 13.8311, Z -1.3333, A 0.000, B 0.000, C 0.000 }
gfCNCPoint1[12705] = {X 301.5523, Y 12.9779, Z -1.3333, A 0.000, B 0.000, C 0.000 }
gfCNCPoint1[12706] = {X 301.5523, Y 12.1868, Z -1.3333, A 0.000, B 0.000, C 0.000 }
gfCNCPoint1[12707] = {X 301.6525, Y 11.2967, Z -1.3333, A 0.000, B 0.000, C 0.000 }
gfCNCPoint1[12708] = {X 301.9484, Y 10.4513, Z -1.3333, A 0.000, B 0.000, C 0.000 }
gfCNCPoint1[12709] = {X 302.4249, Y 9.6929, Z -1.3333, A 0.000, B 0.000, C 0.000 }
gfCNCPoint1[12710] = {X 303.0583, Y 9.0595, Z -1.3333, A 0.000, B 0.000, C 0.000 }
gfCNCPoint1[12711] = {X 303.8167, Y 8.5829, Z -1.3333, A 0.000, B 0.000, C 0.000 }
gfCNCPoint1[12712] = {X 304.6622, Y 8.2871, Z -1.3333, A 0.000, B 0.000, C 0.000 }
gfCNCPoint1[12713] = {X 305.5523, Y 8.1868, Z -1.3333, A 0.000, B 0.000, C 0.000 }
gfCNCPoint1[12714] = {X 311.9957, Y 8.1868, Z -1.3333, A 0.000, B 0.000, C 0.000 }
gfCNCPoint1[12715] = {X 312.8858, Y 8.2871, Z -1.3333, A 0.000, B 0.000, C 0.000 }
gfCNCPoint1[12716] = {X 313.7313, Y 8.5829, Z -1.3333, A 0.000, B 0.000, C 0.000 }
gfCNCPoint1[12717] = {X 314.4897, Y 9.0595, Z -1.3333, A 0.000, B 0.000, C 0.000 }
gfCNCPoint1[12718] = {X 315.1230, Y 9.6929, Z -1.3333, A 0.000, B 0.000, C 0.000 }
gfCNCPoint1[12719] = {X 315.5996, Y 10.4513, Z -1.3333, A 0.000, B 0.000, C 0.000 }
gfCNCPoint1[12720] = {X 315.8954, Y 11.2967, Z -1.3333, A 0.000, B 0.000, C 0.000 }
gfCNCPoint1[12721] = {X 315.9957, Y 12.1868, Z -1.3333, A 0.000, B 0.000, C 0.000 }
gfCNCPoint1[12722] = {X 315.9955, Y 13.0192, Z -1.3333, A 0.000, B 0.000, C 0.000 }
gfCNCPoint1[12723] = {X 315.8970, Y 13.8614, Z -1.3333, A 0.000, B 0.000, C 0.000 }
gfCNCPoint1[12724] = {X 315.6231, Y 14.6638, Z -1.3333, A 0.000, B 0.000, C 0.000 }
gfCNCPoint1[12725] = {X 315.1863, Y 15.3905, Z -1.3333, A 0.000, B 0.000, C 0.000 }
gfCNCPoint1[12726] = {X 314.6061, Y 16.0088, Z -1.3333, A 0.000, B 0.000, C 0.000 }
gfCNCPoint1[12727] = {X 314.5384, Y 16.0658, Z -1.3333, A 0.000, B 0.000, C 0.000 }
gfCNCPoint1[12728] = {X 314.4695, Y 16.1213, Z -1.3333, A 0.000, B 0.000, C 0.000 }
gfCNCPoint1[12729] = {X 314.4671, Y 16.3119, Z -1.3333, A 0.000, B 0.000, C 0.000 }
gfCNCPoint1[12730] = {X 314.4669, Y 41.0670, Z -1.3333, A 0.000, B 0.000, C 0.000 }
gfCNCPoint1[12731] = {X 314.6059, Y 41.1778, Z -1.3333, A 0.000, B 0.000, C 0.000 }
gfCNCPoint1[12732] = {X 315.1924, Y 41.8043, Z -1.3333, A 0.000, B 0.000, C 0.000 }
gfCNCPoint1[12733] = {X 315.6317, Y 42.5416, Z -1.3333, A 0.000, B 0.000, C 0.000 }
gfCNCPoint1[12734] = {X 315.9037, Y 43.3556, Z -1.3333, A 0.000, B 0.000, C 0.000 }
gfCNCPoint1[12735] = {X 315.9957, Y 44.2089, Z -1.3333, A 0.000, B 0.000, C 0.000 }
gfCNCPoint1[12736] = {X 315.9957, Y 45.0000, Z -1.3333, A 0.000, B 0.000, C 0.000 }
gfCNCPoint1[12737] = {X 315.8954, Y 45.8901, Z -1.3333, A 0.000, B 0.000, C 0.000 }
gfCNCPoint1[12738] = {X 315.5996, Y 46.7355, Z -1.3333, A 0.000, B 0.000, C 0.000 }
gfCNCPoint1[12739] = {X 315.1230, Y 47.4940, Z -1.3333, A 0.000, B 0.000, C 0.000 }
gfCNCPoint1[12740] = {X 314.4897, Y 48.1273, Z -1.3333, A 0.000, B 0.000, C 0.000 }
gfCNCPoint1[12741] = {X 313.7313, Y 48.6039, Z -1.3333, A 0.000, B 0.000, C 0.000 }
gfCNCPoint1[12742] = {X 312.8858, Y 48.8997, Z -1.3333, A 0.000, B 0.000, C 0.000 }
gfCNCPoint1[12743] = {X 311.9957, Y 49.0000, Z -1.3333, A 0.000, B 0.000, C 0.000 }
gfCNCPoint1[12744] = {X 305.5523, Y 49.0000, Z -1.3333, A 0.000, B 0.000, C 0.000 }
gfCNCPoint1[12745] = {X 304.6622, Y 48.8997, Z -1.3333, A 0.000, B 0.000, C 0.000 }
gfCNCPoint1[12746] = {X 303.8167, Y 48.6039, Z -1.3333, A 0.000, B 0.000, C 0.000 }
gfCNCPoint1[12747] = {X 303.0583, Y 48.1273, Z -1.3333, A 0.000, B 0.000, C 0.000 }
gfCNCPoint1[12748] = {X 302.4249, Y 47.4939, Z -1.3333, A 0.000, B 0.000, C 0.000 }
gfCNCPoint1[12749] = {X 301.9484, Y 46.7355, Z -1.3333, A 0.000, B 0.000, C 0.000 }
gfCNCPoint1[12750] = {X 301.6525, Y 45.8900, Z -1.3333, A 0.000, B 0.000, C 0.000 }
gfCNCPoint1[12751] = {X 301.5523, Y 44.9999, Z -1.3333, A 0.000, B 0.000, C 0.000 }
gfCNCPoint1[12752] = {X 301.5523, Y 44.2089, Z -1.3333, A 0.000, B 0.000, C 0.000 }
gfCNCPoint1[12753] = {X 301.6704, Y 43.3030, Z -1.3333, A 0.000, B 0.000, C 0.000 }
gfCNCPoint1[12754] = {X 301.9747, Y 42.4415, Z -1.3333, A 0.000, B 0.000, C 0.000 }
gfCNCPoint1[12755] = {X 302.4520, Y 41.6624, Z -1.3333, A 0.000, B 0.000, C 0.000 }
gfCNCPoint1[12756] = {X 303.0811, Y 40.9999, Z -1.3333, A 0.000, B 0.000, C 0.000 }
gfCNCPoint1[12757] = {X 303.0811, Y 33.7143, Z -1.3333, A 0.000, B 0.000, C 0.000 }
gfCNCPoint1[12758] = {X 293.9335, Y 33.7143, Z -1.3333, A 0.000, B 0.000, C 0.000 }
gfCNCPoint1[12759] = {X 293.5336, Y 33.7129, Z -1.3333, A 0.000, B 0.000, C 0.000 }
gfCNCPoint1[12760] = {X 293.5324, Y 41.0525, Z -1.3333, A 0.000, B 0.000, C 0.000 }
gfCNCPoint1[12761] = {X 294.1697, Y 41.6939, Z -1.3333, A 0.000, B 0.000, C 0.000 }
gfCNCPoint1[12762] = {X 294.6510, Y 42.4592, Z -1.3333, A 0.000, B 0.000, C 0.000 }
gfCNCPoint1[12763] = {X 294.9530, Y 43.3113, Z -1.3333, A 0.000, B 0.000, C 0.000 }
gfCNCPoint1[12764] = {X 295.0611, Y 44.2089, Z -1.3333, A 0.000, B 0.000, C 0.000 }
gfCNCPoint1[12765] = {X 295.0611, Y 45.0000, Z -1.3333, A 0.000, B 0.000, C 0.000 }
gfCNCPoint1[12766] = {X 294.9608, Y 45.8901, Z -1.3333, A 0.000, B 0.000, C 0.000 }
gfCNCPoint1[12767] = {X 294.6650, Y 46.7355, Z -1.3333, A 0.000, B 0.000, C 0.000 }
gfCNCPoint1[12768] = {X 294.1885, Y 47.4940, Z -1.3333, A 0.000, B 0.000, C 0.000 }
gfCNCPoint1[12769] = {X 293.5551, Y 48.1273, Z -1.3333, A 0.000, B 0.000, C 0.000 }
gfCNCPoint1[12770] = {X 292.7967, Y 48.6039, Z -1.3333, A 0.000, B 0.000, C 0.000 }
gfCNCPoint1[12771] = {X 291.9512, Y 48.8997, Z -1.3333, A 0.000, B 0.000, C 0.000 }
gfCNCPoint1[12772] = {X 291.0611, Y 49.0000, Z -1.3333, A 0.000, B 0.000, C 0.000 }
gfCNCPoint1[12773] = {X 284.6177, Y 49.0000, Z -1.3333, A 0.000, B 0.000, C 0.000 }
gfCNCPoint1[12774] = {X 283.7276, Y 48.8997, Z -1.3333, A 0.000, B 0.000, C 0.000 }
gfCNCPoint1[12775] = {X 282.8821, Y 48.6039, Z -1.3333, A 0.000, B 0.000, C 0.000 }
gfCNCPoint1[12776] = {X 282.1237, Y 48.1273, Z -1.3333, A 0.000, B 0.000, C 0.000 }
gfCNCPoint1[12777] = {X 281.4903, Y 47.4939, Z -1.3333, A 0.000, B 0.000, C 0.000 }
gfCNCPoint1[12778] = {X 281.0138, Y 46.7355, Z -1.3333, A 0.000, B 0.000, C 0.000 }
gfCNCPoint1[12779] = {X 280.7179, Y 45.8900, Z -1.3333, A 0.000, B 0.000, C 0.000 }
gfCNCPoint1[12780] = {X 280.6177, Y 45.0000, Z -1.3333, A 0.000, B 0.000, C 0.000 }
gfCNCPoint1[12781] = {X 280.6177, Y 44.2089, Z -1.3333, A 0.000, B 0.000, C 0.000 }
gfCNCPoint1[12782] = {X 280.7236, Y 43.3127, Z -1.3333, A 0.000, B 0.000, C 0.000 }
gfCNCPoint1[12783] = {X 281.0252, Y 42.4621, Z -1.3333, A 0.000, B 0.000, C 0.000 }
gfCNCPoint1[12784] = {X 281.5075, Y 41.6994, Z -1.3333, A 0.000, B 0.000, C 0.000 }
gfCNCPoint1[12785] = {X 282.1465, Y 41.0622, Z -1.3333, A 0.000, B 0.000, C 0.000 }
gfCNCPoint1[12786] = {X 282.1463, Y 28.5932, Z -1.3333, A 0.000, B 0.000, C 0.000 }
gfCNCPoint1[12787] = {X 278.0663, Y 28.5933, Z -1.3333, A 0.000, B 0.000, C 0.000 }
gfCNCPoint1[12788] = {X 278.0663, Y 28.5933, Z 1.6667, A 0.000, B 0.000, C 0.000 }
gfCNCPoint1[12789] = {X 278.0663, Y 28.5933, Z 11.0000, A 0.000, B 0.000, C 0.000 }
gfCNCPoint1[12790] = {X 353.3543, Y 107.0423, Z 11.0000, A 0.000, B 0.000, C 0.000 }
gfCNCPoint1[12791] = {X 353.3543, Y 107.0423, Z 1.6667, A 0.000, B 0.000, C 0.000 }
gfCNCPoint1[12792] = {X 353.3543, Y 107.0423, Z -1.3333, A 0.000, B 0.000, C 0.000 }
gfCNCPoint1[12793] = {X 353.2426, Y 102.9639, Z -1.3333, A 0.000, B 0.000, C 0.000 }
gfCNCPoint1[12794] = {X 347.7204, Y 103.0324, Z -1.3333, A 0.000, B 0.000, C 0.000 }
gfCNCPoint1[12795] = {X 342.1986, Y 102.9357, Z -1.3333, A 0.000, B 0.000, C 0.000 }
gfCNCPoint1[12796] = {X 336.6821, Y 102.6738, Z -1.3333, A 0.000, B 0.000, C 0.000 }
gfCNCPoint1[12797] = {X 333.1922, Y 102.3988, Z -1.3333, A 0.000, B 0.000, C 0.000 }
gfCNCPoint1[12798] = {X 329.7159, Y 101.9858, Z -1.3333, A 0.000, B 0.000, C 0.000 }
gfCNCPoint1[12799] = {X 326.2586, Y 101.4356, Z -1.3333, A 0.000, B 0.000, C 0.000 }
gfCNCPoint1[12800] = {X 323.4092, Y 100.8312, Z -1.3333, A 0.000, B 0.000, C 0.000 }
gfCNCPoint1[12801] = {X 320.6120, Y 100.0183, Z -1.3333, A 0.000, B 0.000, C 0.000 }
gfCNCPoint1[12802] = {X 317.8824, Y 99.0013, Z -1.3333, A 0.000, B 0.000, C 0.000 }
gfCNCPoint1[12803] = {X 316.3691, Y 98.3041, Z -1.3333, A 0.000, B 0.000, C 0.000 }
gfCNCPoint1[12804] = {X 314.9196, Y 97.4824, Z -1.3333, A 0.000, B 0.000, C 0.000 }
gfCNCPoint1[12805] = {X 313.5442, Y 96.5421, Z -1.3333, A 0.000, B 0.000, C 0.000 }
gfCNCPoint1[12806] = {X 312.2525, Y 95.4896, Z -1.3333, A 0.000, B 0.000, C 0.000 }
gfCNCPoint1[12807] = {X 311.2494, Y 94.4912, Z -1.3333, A 0.000, B 0.000, C 0.000 }
gfCNCPoint1[12808] = {X 310.3715, Y 93.3810, Z -1.3333, A 0.000, B 0.000, C 0.000 }
gfCNCPoint1[12809] = {X 309.6314, Y 92.1746, Z -1.3333, A 0.000, B 0.000, C 0.000 }
gfCNCPoint1[12810] = {X 309.0395, Y 90.8890, Z -1.3333, A 0.000, B 0.000, C 0.000 }
gfCNCPoint1[12811] = {X 308.6040, Y 89.5423, Z -1.3333, A 0.000, B 0.000, C 0.000 }
gfCNCPoint1[12812] = {X 308.2605, Y 87.9191, Z -1.3333, A 0.000, B 0.000, C 0.000 }
gfCNCPoint1[12813] = {X 308.0576, Y 86.2725, Z -1.3333, A 0.000, B 0.000, C 0.000 }
gfCNCPoint1[12814] = {X 307.9967, Y 84.6144, Z -1.3333, A 0.000, B 0.000, C 0.000 }
gfCNCPoint1[12815] = {X 307.9980, Y 83.2310, Z -1.3333, A 0.000, B 0.000, C 0.000 }
gfCNCPoint1[12816] = {X 307.9980, Y 63.2124, Z -1.3333, A 0.000, B 0.000, C 0.000 }
gfCNCPoint1[12817] = {X 307.1462, Y 63.0034, Z -1.3333, A 0.000, B 0.000, C 0.000 }
gfCNCPoint1[12818] = {X 306.3542, Y 62.6267, Z -1.3333, A 0.000, B 0.000, C 0.000 }
gfCNCPoint1[12819] = {X 305.6546, Y 62.0978, Z -1.3333, A 0.000, B 0.000, C 0.000 }
gfCNCPoint1[12820] = {X 305.0763, Y 61.4385, Z -1.3333, A 0.000, B 0.000, C 0.000 }
gfCNCPoint1[12821] = {X 304.6430, Y 60.6760, Z -1.3333, A 0.000, B 0.000, C 0.000 }
gfCNCPoint1[12822] = {X 304.3726, Y 59.8417, Z -1.3333, A 0.000, B 0.000, C 0.000 }
gfCNCPoint1[12823] = {X 304.2764, Y 58.9699, Z -1.3333, A 0.000, B 0.000, C 0.000 }
gfCNCPoint1[12824] = {X 304.2762, Y 58.0000, Z -1.3333, A 0.000, B 0.000, C 0.000 }
gfCNCPoint1[12825] = {X 304.3845, Y 57.0387, Z -1.3333, A 0.000, B 0.000, C 0.000 }
gfCNCPoint1[12826] = {X 304.7040, Y 56.1256, Z -1.3333, A 0.000, B 0.000, C 0.000 }
gfCNCPoint1[12827] = {X 305.2187, Y 55.3065, Z -1.3333, A 0.000, B 0.000, C 0.000 }
gfCNCPoint1[12828] = {X 305.9027, Y 54.6225, Z -1.3333, A 0.000, B 0.000, C 0.000 }
gfCNCPoint1[12829] = {X 306.7218, Y 54.1078, Z -1.3333, A 0.000, B 0.000, C 0.000 }
gfCNCPoint1[12830] = {X 307.6349, Y 53.7883, Z -1.3333, A 0.000, B 0.000, C 0.000 }
gfCNCPoint1[12831] = {X 308.5962, Y 53.6800, Z -1.3333, A 0.000, B 0.000, C 0.000 }
gfCNCPoint1[12832] = {X 324.3107, Y 53.6800, Z -1.3333, A 0.000, B 0.000, C 0.000 }
gfCNCPoint1[12833] = {X 325.2720, Y 53.7883, Z -1.3333, A 0.000, B 0.000, C 0.000 }
gfCNCPoint1[12834] = {X 326.1851, Y 54.1078, Z -1.3333, A 0.000, B 0.000, C 0.000 }
gfCNCPoint1[12835] = {X 327.0042, Y 54.6225, Z -1.3333, A 0.000, B 0.000, C 0.000 }
gfCNCPoint1[12836] = {X 327.6882, Y 55.3065, Z -1.3333, A 0.000, B 0.000, C 0.000 }
gfCNCPoint1[12837] = {X 328.2029, Y 56.1256, Z -1.3333, A 0.000, B 0.000, C 0.000 }
gfCNCPoint1[12838] = {X 328.5224, Y 57.0387, Z -1.3333, A 0.000, B 0.000, C 0.000 }
gfCNCPoint1[12839] = {X 328.6307, Y 58.0000, Z -1.3333, A 0.000, B 0.000, C 0.000 }
gfCNCPoint1[12840] = {X 328.6307, Y 58.9361, Z -1.3333, A 0.000, B 0.000, C 0.000 }
gfCNCPoint1[12841] = {X 328.5361, Y 59.8122, Z -1.3333, A 0.000, B 0.000, C 0.000 }
gfCNCPoint1[12842] = {X 328.2673, Y 60.6515, Z -1.3333, A 0.000, B 0.000, C 0.000 }
gfCNCPoint1[12843] = {X 327.8352, Y 61.4195, Z -1.3333, A 0.000, B 0.000, C 0.000 }
gfCNCPoint1[12844] = {X 327.2575, Y 62.0849, Z -1.3333, A 0.000, B 0.000, C 0.000 }
gfCNCPoint1[12845] = {X 326.5578, Y 62.6206, Z -1.3333, A 0.000, B 0.000, C 0.000 }
gfCNCPoint1[12846] = {X 325.7647, Y 63.0047, Z -1.3333, A 0.000, B 0.000, C 0.000 }
gfCNCPoint1[12847] = {X 324.9105, Y 63.2214, Z -1.3333, A 0.000, B 0.000, C 0.000 }
gfCNCPoint1[12848] = {X 324.9119, Y 83.2296, Z -1.3333, A 0.000, B 0.000, C 0.000 }
gfCNCPoint1[12849] = {X 324.9254, Y 84.6149, Z -1.3333, A 0.000, B 0.000, C 0.000 }
gfCNCPoint1[12850] = {X 325.0027, Y 85.8503, Z -1.3333, A 0.000, B 0.000, C 0.000 }
gfCNCPoint1[12851] = {X 325.2260, Y 87.0678, Z -1.3333, A 0.000, B 0.000, C 0.000 }
gfCNCPoint1[12852] = {X 325.4714, Y 87.3369, Z -1.3333, A 0.000, B 0.000, C 0.000 }
gfCNCPoint1[12853] = {X 325.7737, Y 87.5402, Z -1.3333, A 0.000, B 0.000, C 0.000 }
gfCNCPoint1[12854] = {X 326.2232, Y 87.7937, Z -1.3333, A 0.000, B 0.000, C 0.000 }
gfCNCPoint1[12855] = {X 327.6615, Y 88.3915, Z -1.3333, A 0.000, B 0.000, C 0.000 }
gfCNCPoint1[12856] = {X 329.1568, Y 88.8273, Z -1.3333, A 0.000, B 0.000, C 0.000 }
gfCNCPoint1[12857] = {X 332.2328, Y 89.4432, Z -1.3333, A 0.000, B 0.000, C 0.000 }
gfCNCPoint1[12858] = {X 335.3452, Y 89.8355, Z -1.3333, A 0.000, B 0.000, C 0.000 }
gfCNCPoint1[12859] = {X 340.5196, Y 90.2185, Z -1.3333, A 0.000, B 0.000, C 0.000 }
gfCNCPoint1[12860] = {X 345.7061, Y 90.3632, Z -1.3333, A 0.000, B 0.000, C 0.000 }
gfCNCPoint1[12861] = {X 350.5483, Y 90.3692, Z -1.3333, A 0.000, B 0.000, C 0.000 }
gfCNCPoint1[12862] = {X 355.3876, Y 90.2008, Z -1.3333, A 0.000, B 0.000, C 0.000 }
gfCNCPoint1[12863] = {X 360.2177, Y 89.8581, Z -1.3333, A 0.000, B 0.000, C 0.000 }
gfCNCPoint1[12864] = {X 362.7645, Y 89.5689, Z -1.3333, A 0.000, B 0.000, C 0.000 }
gfCNCPoint1[12865] = {X 365.2878, Y 89.1188, Z -1.3333, A 0.000, B 0.000, C 0.000 }
gfCNCPoint1[12866] = {X 367.7776, Y 88.5096, Z -1.3333, A 0.000, B 0.000, C 0.000 }
gfCNCPoint1[12867] = {X 368.7096, Y 88.1962, Z -1.3333, A 0.000, B 0.000, C 0.000 }
gfCNCPoint1[12868] = {X 369.6005, Y 87.7803, Z -1.3333, A 0.000, B 0.000, C 0.000 }
gfCNCPoint1[12869] = {X 370.4392, Y 87.2670, Z -1.3333, A 0.000, B 0.000, C 0.000 }
gfCNCPoint1[12870] = {X 370.5892, Y 87.1109, Z -1.3333, A 0.000, B 0.000, C 0.000 }
gfCNCPoint1[12871] = {X 370.6666, Y 86.9086, Z -1.3333, A 0.000, B 0.000, C 0.000 }
gfCNCPoint1[12872] = {X 370.8577, Y 85.3734, Z -1.3333, A 0.000, B 0.000, C 0.000 }
gfCNCPoint1[12873] = {X 370.9214, Y 83.8276, Z -1.3333, A 0.000, B 0.000, C 0.000 }
gfCNCPoint1[12874] = {X 370.9211, Y 63.2125, Z -1.3333, A 0.000, B 0.000, C 0.000 }
gfCNCPoint1[12875] = {X 370.0693, Y 63.0035, Z -1.3333, A 0.000, B 0.000, C 0.000 }
gfCNCPoint1[12876] = {X 369.2773, Y 62.6267, Z -1.3333, A 0.000, B 0.000, C 0.000 }
gfCNCPoint1[12877] = {X 368.5777, Y 62.0978, Z -1.3333, A 0.000, B 0.000, C 0.000 }
gfCNCPoint1[12878] = {X 367.9993, Y 61.4385, Z -1.3333, A 0.000, B 0.000, C 0.000 }
gfCNCPoint1[12879] = {X 367.5660, Y 60.6759, Z -1.3333, A 0.000, B 0.000, C 0.000 }
gfCNCPoint1[12880] = {X 367.2957, Y 59.8415, Z -1.3333, A 0.000, B 0.000, C 0.000 }
gfCNCPoint1[12881] = {X 367.1994, Y 58.9697, Z -1.3333, A 0.000, B 0.000, C 0.000 }
gfCNCPoint1[12882] = {X 367.1993, Y 58.0000, Z -1.3333, A 0.000, B 0.000, C 0.000 }
gfCNCPoint1[12883] = {X 367.3076, Y 57.0387, Z -1.3333, A 0.000, B 0.000, C 0.000 }
gfCNCPoint1[12884] = {X 367.6271, Y 56.1256, Z -1.3333, A 0.000, B 0.000, C 0.000 }
gfCNCPoint1[12885] = {X 368.1418, Y 55.3065, Z -1.3333, A 0.000, B 0.000, C 0.000 }
gfCNCPoint1[12886] = {X 368.8258, Y 54.6225, Z -1.3333, A 0.000, B 0.000, C 0.000 }
gfCNCPoint1[12887] = {X 369.6449, Y 54.1078, Z -1.3333, A 0.000, B 0.000, C 0.000 }
gfCNCPoint1[12888] = {X 370.5580, Y 53.7883, Z -1.3333, A 0.000, B 0.000, C 0.000 }
gfCNCPoint1[12889] = {X 371.5193, Y 53.6800, Z -1.3333, A 0.000, B 0.000, C 0.000 }
gfCNCPoint1[12890] = {X 388.0597, Y 53.6800, Z -1.3333, A 0.000, B 0.000, C 0.000 }
gfCNCPoint1[12891] = {X 389.0210, Y 53.7883, Z -1.3333, A 0.000, B 0.000, C 0.000 }
gfCNCPoint1[12892] = {X 389.9341, Y 54.1078, Z -1.3333, A 0.000, B 0.000, C 0.000 }
gfCNCPoint1[12893] = {X 390.7532, Y 54.6225, Z -1.3333, A 0.000, B 0.000, C 0.000 }
gfCNCPoint1[12894] = {X 391.4372, Y 55.3065, Z -1.3333, A 0.000, B 0.000, C 0.000 }
gfCNCPoint1[12895] = {X 391.9519, Y 56.1256, Z -1.3333, A 0.000, B 0.000, C 0.000 }
gfCNCPoint1[12896] = {X 392.2714, Y 57.0387, Z -1.3333, A 0.000, B 0.000, C 0.000 }
gfCNCPoint1[12897] = {X 392.3797, Y 58.0000, Z -1.3333, A 0.000, B 0.000, C 0.000 }
gfCNCPoint1[12898] = {X 392.3797, Y 58.9342, Z -1.3333, A 0.000, B 0.000, C 0.000 }
gfCNCPoint1[12899] = {X 392.2634, Y 59.9297, Z -1.3333, A 0.000, B 0.000, C 0.000 }
gfCNCPoint1[12900] = {X 391.9209, Y 60.8715, Z -1.3333, A 0.000, B 0.000, C 0.000 }
gfCNCPoint1[12901] = {X 391.4769, Y 61.5794, Z -1.3333, A 0.000, B 0.000, C 0.000 }
gfCNCPoint1[12902] = {X 390.9056, Y 62.1890, Z -1.3333, A 0.000, B 0.000, C 0.000 }
gfCNCPoint1[12903] = {X 390.2280, Y 62.6779, Z -1.3333, A 0.000, B 0.000, C 0.000 }
gfCNCPoint1[12904] = {X 389.4693, Y 63.0279, Z -1.3333, A 0.000, B 0.000, C 0.000 }
gfCNCPoint1[12905] = {X 388.6576, Y 63.2261, Z -1.3333, A 0.000, B 0.000, C 0.000 }
gfCNCPoint1[12906] = {X 388.6556, Y 84.6147, Z -1.3333, A 0.000, B 0.000, C 0.000 }
gfCNCPoint1[12907] = {X 388.5955, Y 86.2731, Z -1.3333, A 0.000, B 0.000, C 0.000 }
gfCNCPoint1[12908] = {X 388.3912, Y 87.9199, Z -1.3333, A 0.000, B 0.000, C 0.000 }
gfCNCPoint1[12909] = {X 388.0441, Y 89.5426, Z -1.3333, A 0.000, B 0.000, C 0.000 }
gfCNCPoint1[12910] = {X 387.5121, Y 91.1300, Z -1.3333, A 0.000, B 0.000, C 0.000 }
gfCNCPoint1[12911] = {X 386.7626, Y 92.6270, Z -1.3333, A 0.000, B 0.000, C 0.000 }
gfCNCPoint1[12912] = {X 385.8104, Y 94.0040, Z -1.3333, A 0.000, B 0.000, C 0.000 }
gfCNCPoint1[12913] = {X 384.6745, Y 95.2338, Z -1.3333, A 0.000, B 0.000, C 0.000 }
gfCNCPoint1[12914] = {X 383.1604, Y 96.5092, Z -1.3333, A 0.000, B 0.000, C 0.000 }
gfCNCPoint1[12915] = {X 381.5196, Y 97.6168, Z -1.3333, A 0.000, B 0.000, C 0.000 }
gfCNCPoint1[12916] = {X 379.7706, Y 98.5441, Z -1.3333, A 0.000, B 0.000, C 0.000 }
gfCNCPoint1[12917] = {X 377.4996, Y 99.5015, Z -1.3333, A 0.000, B 0.000, C 0.000 }
gfCNCPoint1[12918] = {X 375.1653, Y 100.2918, Z -1.3333, A 0.000, B 0.000, C 0.000 }
gfCNCPoint1[12919] = {X 372.7799, Y 100.9110, Z -1.3333, A 0.000, B 0.000, C 0.000 }
gfCNCPoint1[12920] = {X 368.9683, Y 101.6484, Z -1.3333, A 0.000, B 0.000, C 0.000 }
gfCNCPoint1[12921] = {X 365.1256, Y 102.2018, Z -1.3333, A 0.000, B 0.000, C 0.000 }
gfCNCPoint1[12922] = {X 361.2608, Y 102.5697, Z -1.3333, A 0.000, B 0.000, C 0.000 }
gfCNCPoint1[12923] = {X 357.2539, Y 102.8104, Z -1.3333, A 0.000, B 0.000, C 0.000 }
gfCNCPoint1[12924] = {X 353.2426, Y 102.9639, Z -1.3333, A 0.000, B 0.000, C 0.000 }
gfCNCPoint1[12925] = {X 353.3521, Y 106.9624, Z -1.3333, A 0.000, B 0.000, C 0.000 }
gfCNCPoint1[12926] = {X 353.2404, Y 102.8839, Z -1.3333, A 0.000, B 0.000, C 0.000 }
gfCNCPoint1[12927] = {X 347.7205, Y 102.9524, Z -1.3333, A 0.000, B 0.000, C 0.000 }
gfCNCPoint1[12928] = {X 342.2011, Y 102.8557, Z -1.3333, A 0.000, B 0.000, C 0.000 }
gfCNCPoint1[12929] = {X 336.6870, Y 102.5939, Z -1.3333, A 0.000, B 0.000, C 0.000 }
gfCNCPoint1[12930] = {X 333.2001, Y 102.3192, Z -1.3333, A 0.000, B 0.000, C 0.000 }
gfCNCPoint1[12931] = {X 329.7268, Y 101.9066, Z -1.3333, A 0.000, B 0.000, C 0.000 }
gfCNCPoint1[12932] = {X 326.2726, Y 101.3568, Z -1.3333, A 0.000, B 0.000, C 0.000 }
gfCNCPoint1[12933] = {X 323.4288, Y 100.7536, Z -1.3333, A 0.000, B 0.000, C 0.000 }
gfCNCPoint1[12934] = {X 320.6371, Y 99.9423, Z -1.3333, A 0.000, B 0.000, C 0.000 }
gfCNCPoint1[12935] = {X 317.9129, Y 98.9274, Z -1.3333, A 0.000, B 0.000, C 0.000 }
gfCNCPoint1[12936] = {X 316.4057, Y 98.2330, Z -1.3333, A 0.000, B 0.000, C 0.000 }
gfCNCPoint1[12937] = {X 314.9620, Y 97.4146, Z -1.3333, A 0.000, B 0.000, C 0.000 }
gfCNCPoint1[12938] = {X 313.5921, Y 96.4780, Z -1.3333, A 0.000, B 0.000, C 0.000 }
gfCNCPoint1[12939] = {X 312.3056, Y 95.4297, Z -1.3333, A 0.000, B 0.000, C 0.000 }
gfCNCPoint1[12940] = {X 311.3091, Y 94.4380, Z -1.3333, A 0.000, B 0.000, C 0.000 }
gfCNCPoint1[12941] = {X 310.4372, Y 93.3352, Z -1.3333, A 0.000, B 0.000, C 0.000 }
gfCNCPoint1[12942] = {X 309.7020, Y 92.1369, Z -1.3333, A 0.000, B 0.000, C 0.000 }
gfCNCPoint1[12943] = {X 309.1140, Y 90.8599, Z -1.3333, A 0.000, B 0.000, C 0.000 }
gfCNCPoint1[12944] = {X 308.6814, Y 89.5223, Z -1.3333, A 0.000, B 0.000, C 0.000 }
gfCNCPoint1[12945] = {X 308.3394, Y 87.9058, Z -1.3333, A 0.000, B 0.000, C 0.000 }
gfCNCPoint1[12946] = {X 308.1373, Y 86.2660, Z -1.3333, A 0.000, B 0.000, C 0.000 }
gfCNCPoint1[12947] = {X 308.0767, Y 84.6148, Z -1.3333, A 0.000, B 0.000, C 0.000 }
gfCNCPoint1[12948] = {X 308.0780, Y 83.2310, Z -1.3333, A 0.000, B 0.000, C 0.000 }
gfCNCPoint1[12949] = {X 308.0780, Y 63.1423, Z -1.3333, A 0.000, B 0.000, C 0.000 }
gfCNCPoint1[12950] = {X 307.2293, Y 62.9477, Z -1.3333, A 0.000, B 0.000, C 0.000 }
gfCNCPoint1[12951] = {X 306.4383, Y 62.5839, Z -1.3333, A 0.000, B 0.000, C 0.000 }
gfCNCPoint1[12952] = {X 305.7383, Y 62.0661, Z -1.3333, A 0.000, B 0.000, C 0.000 }
gfCNCPoint1[12953] = {X 305.1588, Y 61.4164, Z -1.3333, A 0.000, B 0.000, C 0.000 }
gfCNCPoint1[12954] = {X 304.7242, Y 60.6619, Z -1.3333, A 0.000, B 0.000, C 0.000 }
gfCNCPoint1[12955] = {X 304.4530, Y 59.8346, Z -1.3333, A 0.000, B 0.000, C 0.000 }
gfCNCPoint1[12956] = {X 304.3564, Y 58.9693, Z -1.3333, A 0.000, B 0.000, C 0.000 }
gfCNCPoint1[12957] = {X 304.3562, Y 58.0000, Z -1.3333, A 0.000, B 0.000, C 0.000 }
gfCNCPoint1[12958] = {X 304.4625, Y 57.0565, Z -1.3333, A 0.000, B 0.000, C 0.000 }
gfCNCPoint1[12959] = {X 304.7761, Y 56.1603, Z -1.3333, A 0.000, B 0.000, C 0.000 }
gfCNCPoint1[12960] = {X 305.2813, Y 55.3564, Z -1.3333, A 0.000, B 0.000, C 0.000 }
gfCNCPoint1[12961] = {X 305.9526, Y 54.6850, Z -1.3333, A 0.000, B 0.000, C 0.000 }
gfCNCPoint1[12962] = {X 306.7566, Y 54.1799, Z -1.3333, A 0.000, B 0.000, C 0.000 }
gfCNCPoint1[12963] = {X 307.6527, Y 53.8663, Z -1.3333, A 0.000, B 0.000, C 0.000 }
gfCNCPoint1[12964] = {X 308.5962, Y 53.7600, Z -1.3333, A 0.000, B 0.000, C 0.000 }
gfCNCPoint1[12965] = {X 324.3107, Y 53.7600, Z -1.3333, A 0.000, B 0.000, C 0.000 }
gfCNCPoint1[12966] = {X 325.2542, Y 53.8663, Z -1.3333, A 0.000, B 0.000, C 0.000 }
gfCNCPoint1[12967] = {X 326.1504, Y 54.1799, Z -1.3333, A 0.000, B 0.000, C 0.000 }
gfCNCPoint1[12968] = {X 326.9543, Y 54.6850, Z -1.3333, A 0.000, B 0.000, C 0.000 }
gfCNCPoint1[12969] = {X 327.6257, Y 55.3564, Z -1.3333, A 0.000, B 0.000, C 0.000 }
gfCNCPoint1[12970] = {X 328.1308, Y 56.1603, Z -1.3333, A 0.000, B 0.000, C 0.000 }
gfCNCPoint1[12971] = {X 328.4444, Y 57.0565, Z -1.3333, A 0.000, B 0.000, C 0.000 }
gfCNCPoint1[12972] = {X 328.5507, Y 58.0000, Z -1.3333, A 0.000, B 0.000, C 0.000 }
gfCNCPoint1[12973] = {X 328.5507, Y 58.9356, Z -1.3333, A 0.000, B 0.000, C 0.000 }
gfCNCPoint1[12974] = {X 328.4558, Y 59.8053, Z -1.3333, A 0.000, B 0.000, C 0.000 }
gfCNCPoint1[12975] = {X 328.1860, Y 60.6375, Z -1.3333, A 0.000, B 0.000, C 0.000 }
gfCNCPoint1[12976] = {X 327.7527, Y 61.3975, Z -1.3333, A 0.000, B 0.000, C 0.000 }
gfCNCPoint1[12977] = {X 327.1739, Y 62.0535, Z -1.3333, A 0.000, B 0.000, C 0.000 }
gfCNCPoint1[12978] = {X 326.4738, Y 62.5781, Z -1.3333, A 0.000, B 0.000, C 0.000 }
gfCNCPoint1[12979] = {X 325.6816, Y 62.9494, Z -1.3333, A 0.000, B 0.000, C 0.000 }
gfCNCPoint1[12980] = {X 324.8305, Y 63.1519, Z -1.3333, A 0.000, B 0.000, C 0.000 }
gfCNCPoint1[12981] = {X 324.8319, Y 83.2300, Z -1.3333, A 0.000, B 0.000, C 0.000 }
gfCNCPoint1[12982] = {X 324.8454, Y 84.6152, Z -1.3333, A 0.000, B 0.000, C 0.000 }
gfCNCPoint1[12983] = {X 324.9243, Y 85.8675, Z -1.3333, A 0.000, B 0.000, C 0.000 }
gfCNCPoint1[12984] = {X 325.1520, Y 87.1016, Z -1.3333, A 0.000, B 0.000, C 0.000 }
gfCNCPoint1[12985] = {X 325.4127, Y 87.3919, Z -1.3333, A 0.000, B 0.000, C 0.000 }
gfCNCPoint1[12986] = {X 325.7358, Y 87.6107, Z -1.3333, A 0.000, B 0.000, C 0.000 }
gfCNCPoint1[12987] = {X 326.1862, Y 87.8647, Z -1.3333, A 0.000, B 0.000, C 0.000 }
gfCNCPoint1[12988] = {X 327.6337, Y 88.4665, Z -1.3333, A 0.000, B 0.000, C 0.000 }
gfCNCPoint1[12989] = {X 329.1387, Y 88.9052, Z -1.3333, A 0.000, B 0.000, C 0.000 }
gfCNCPoint1[12990] = {X 332.2201, Y 89.5222, Z -1.3333, A 0.000, B 0.000, C 0.000 }
gfCNCPoint1[12991] = {X 335.3381, Y 89.9152, Z -1.3333, A 0.000, B 0.000, C 0.000 }
gfCNCPoint1[12992] = {X 340.5158, Y 90.2984, Z -1.3333, A 0.000, B 0.000, C 0.000 }
gfCNCPoint1[12993] = {X 345.7057, Y 90.4432, Z -1.3333, A 0.000, B 0.000, C 0.000 }
gfCNCPoint1[12994] = {X 350.5504, Y 90.4492, Z -1.3333, A 0.000, B 0.000, C 0.000 }
gfCNCPoint1[12995] = {X 355.3922, Y 90.2806, Z -1.3333, A 0.000, B 0.000, C 0.000 }
gfCNCPoint1[12996] = {X 360.2248, Y 89.9378, Z -1.3333, A 0.000, B 0.000, C 0.000 }
gfCNCPoint1[12997] = {X 362.7764, Y 89.6480, Z -1.3333, A 0.000, B 0.000, C 0.000 }
gfCNCPoint1[12998] = {X 365.3046, Y 89.1970, Z -1.3333, A 0.000, B 0.000, C 0.000 }
gfCNCPoint1[12999] = {X 367.7990, Y 88.5867, Z -1.3333, A 0.000, B 0.000, C 0.000 }
gfCNCPoint1[13000] = {X 368.7394, Y 88.2704, Z -1.3333, A 0.000, B 0.000, C 0.000 }
gfCNCPoint1[13001] = {X 369.6385, Y 87.8507, Z -1.3333, A 0.000, B 0.000, C 0.000 }
gfCNCPoint1[13002] = {X 370.4847, Y 87.3328, Z -1.3333, A 0.000, B 0.000, C 0.000 }
gfCNCPoint1[13003] = {X 370.6568, Y 87.1537, Z -1.3333, A 0.000, B 0.000, C 0.000 }
gfCNCPoint1[13004] = {X 370.7455, Y 86.9217, Z -1.3333, A 0.000, B 0.000, C 0.000 }
gfCNCPoint1[13005] = {X 370.9374, Y 85.3800, Z -1.3333, A 0.000, B 0.000, C 0.000 }
gfCNCPoint1[13006] = {X 371.0014, Y 83.8276, Z -1.3333, A 0.000, B 0.000, C 0.000 }
gfCNCPoint1[13007] = {X 371.0011, Y 63.1423, Z -1.3333, A 0.000, B 0.000, C 0.000 }
gfCNCPoint1[13008] = {X 370.1524, Y 62.9477, Z -1.3333, A 0.000, B 0.000, C 0.000 }
gfCNCPoint1[13009] = {X 369.3614, Y 62.5839, Z -1.3333, A 0.000, B 0.000, C 0.000 }
gfCNCPoint1[13010] = {X 368.6613, Y 62.0661, Z -1.3333, A 0.000, B 0.000, C 0.000 }
gfCNCPoint1[13011] = {X 368.0818, Y 61.4163, Z -1.3333, A 0.000, B 0.000, C 0.000 }
gfCNCPoint1[13012] = {X 367.6473, Y 60.6618, Z -1.3333, A 0.000, B 0.000, C 0.000 }
gfCNCPoint1[13013] = {X 367.3760, Y 59.8344, Z -1.3333, A 0.000, B 0.000, C 0.000 }
gfCNCPoint1[13014] = {X 367.2794, Y 58.9691, Z -1.3333, A 0.000, B 0.000, C 0.000 }
gfCNCPoint1[13015] = {X 367.2793, Y 58.0000, Z -1.3333, A 0.000, B 0.000, C 0.000 }
gfCNCPoint1[13016] = {X 367.3856, Y 57.0565, Z -1.3333, A 0.000, B 0.000, C 0.000 }
gfCNCPoint1[13017] = {X 367.6992, Y 56.1603, Z -1.3333, A 0.000, B 0.000, C 0.000 }
gfCNCPoint1[13018] = {X 368.2043, Y 55.3564, Z -1.3333, A 0.000, B 0.000, C 0.000 }
gfCNCPoint1[13019] = {X 368.8757, Y 54.6850, Z -1.3333, A 0.000, B 0.000, C 0.000 }
gfCNCPoint1[13020] = {X 369.6796, Y 54.1799, Z -1.3333, A 0.000, B 0.000, C 0.000 }
gfCNCPoint1[13021] = {X 370.5758, Y 53.8663, Z -1.3333, A 0.000, B 0.000, C 0.000 }
gfCNCPoint1[13022] = {X 371.5193, Y 53.7600, Z -1.3333, A 0.000, B 0.000, C 0.000 }
gfCNCPoint1[13023] = {X 388.0597, Y 53.7600, Z -1.3333, A 0.000, B 0.000, C 0.000 }
gfCNCPoint1[13024] = {X 389.0032, Y 53.8663, Z -1.3333, A 0.000, B 0.000, C 0.000 }
gfCNCPoint1[13025] = {X 389.8993, Y 54.1799, Z -1.3333, A 0.000, B 0.000, C 0.000 }
gfCNCPoint1[13026] = {X 390.7033, Y 54.6850, Z -1.3333, A 0.000, B 0.000, C 0.000 }
gfCNCPoint1[13027] = {X 391.3746, Y 55.3564, Z -1.3333, A 0.000, B 0.000, C 0.000 }
gfCNCPoint1[13028] = {X 391.8798, Y 56.1603, Z -1.3333, A 0.000, B 0.000, C 0.000 }
gfCNCPoint1[13029] = {X 392.1934, Y 57.0565, Z -1.3333, A 0.000, B 0.000, C 0.000 }
gfCNCPoint1[13030] = {X 392.2997, Y 58.0000, Z -1.3333, A 0.000, B 0.000, C 0.000 }
gfCNCPoint1[13031] = {X 392.2997, Y 58.9342, Z -1.3333, A 0.000, B 0.000, C 0.000 }
gfCNCPoint1[13032] = {X 392.1855, Y 59.9112, Z -1.3333, A 0.000, B 0.000, C 0.000 }
gfCNCPoint1[13033] = {X 391.8493, Y 60.8356, Z -1.3333, A 0.000, B 0.000, C 0.000 }
gfCNCPoint1[13034] = {X 391.4051, Y 61.5414, Z -1.3333, A 0.000, B 0.000, C 0.000 }
gfCNCPoint1[13035] = {X 390.8319, Y 62.1471, Z -1.3333, A 0.000, B 0.000, C 0.000 }
gfCNCPoint1[13036] = {X 390.1517, Y 62.6296, Z -1.3333, A 0.000, B 0.000, C 0.000 }
gfCNCPoint1[13037] = {X 389.3906, Y 62.9703, Z -1.3333, A 0.000, B 0.000, C 0.000 }
gfCNCPoint1[13038] = {X 388.5776, Y 63.1562, Z -1.3333, A 0.000, B 0.000, C 0.000 }
gfCNCPoint1[13039] = {X 388.5756, Y 84.6150, Z -1.3333, A 0.000, B 0.000, C 0.000 }
gfCNCPoint1[13040] = {X 388.5158, Y 86.2665, Z -1.3333, A 0.000, B 0.000, C 0.000 }
gfCNCPoint1[13041] = {X 388.3123, Y 87.9065, Z -1.3333, A 0.000, B 0.000, C 0.000 }
gfCNCPoint1[13042] = {X 387.9667, Y 89.5225, Z -1.3333, A 0.000, B 0.000, C 0.000 }
gfCNCPoint1[13043] = {X 387.4382, Y 91.0992, Z -1.3333, A 0.000, B 0.000, C 0.000 }
gfCNCPoint1[13044] = {X 386.6938, Y 92.5862, Z -1.3333, A 0.000, B 0.000, C 0.000 }
gfCNCPoint1[13045] = {X 385.7480, Y 93.9540, Z -1.3333, A 0.000, B 0.000, C 0.000 }
gfCNCPoint1[13046] = {X 384.6197, Y 95.1755, Z -1.3333, A 0.000, B 0.000, C 0.000 }
gfCNCPoint1[13047] = {X 383.1121, Y 96.4454, Z -1.3333, A 0.000, B 0.000, C 0.000 }
gfCNCPoint1[13048] = {X 381.4784, Y 97.5483, Z -1.3333, A 0.000, B 0.000, C 0.000 }
gfCNCPoint1[13049] = {X 379.7368, Y 98.4716, Z -1.3333, A 0.000, B 0.000, C 0.000 }
gfCNCPoint1[13050] = {X 377.4713, Y 99.4267, Z -1.3333, A 0.000, B 0.000, C 0.000 }
gfCNCPoint1[13051] = {X 375.1425, Y 100.2151, Z -1.3333, A 0.000, B 0.000, C 0.000 }
gfCNCPoint1[13052] = {X 372.7627, Y 100.8329, Z -1.3333, A 0.000, B 0.000, C 0.000 }
gfCNCPoint1[13053] = {X 368.9549, Y 101.5696, Z -1.3333, A 0.000, B 0.000, C 0.000 }
gfCNCPoint1[13054] = {X 365.1161, Y 102.1223, Z -1.3333, A 0.000, B 0.000, C 0.000 }
gfCNCPoint1[13055] = {X 361.2551, Y 102.4899, Z -1.3333, A 0.000, B 0.000, C 0.000 }
gfCNCPoint1[13056] = {X 357.2499, Y 102.7305, Z -1.3333, A 0.000, B 0.000, C 0.000 }
gfCNCPoint1[13057] = {X 353.2404, Y 102.8839, Z -1.3333, A 0.000, B 0.000, C 0.000 }
gfCNCPoint1[13058] = {X 353.3499, Y 106.8824, Z -1.3333, A 0.000, B 0.000, C 0.000 }
gfCNCPoint1[13059] = {X 353.2382, Y 102.8039, Z -1.3333, A 0.000, B 0.000, C 0.000 }
gfCNCPoint1[13060] = {X 347.7207, Y 102.8724, Z -1.3333, A 0.000, B 0.000, C 0.000 }
gfCNCPoint1[13061] = {X 342.2036, Y 102.7757, Z -1.3333, A 0.000, B 0.000, C 0.000 }
gfCNCPoint1[13062] = {X 336.6919, Y 102.5141, Z -1.3333, A 0.000, B 0.000, C 0.000 }
gfCNCPoint1[13063] = {X 333.2080, Y 102.2395, Z -1.3333, A 0.000, B 0.000, C 0.000 }
gfCNCPoint1[13064] = {X 329.7377, Y 101.8273, Z -1.3333, A 0.000, B 0.000, C 0.000 }
gfCNCPoint1[13065] = {X 326.2865, Y 101.2781, Z -1.3333, A 0.000, B 0.000, C 0.000 }
gfCNCPoint1[13066] = {X 323.4483, Y 100.6760, Z -1.3333, A 0.000, B 0.000, C 0.000 }
gfCNCPoint1[13067] = {X 320.6623, Y 99.8664, Z -1.3333, A 0.000, B 0.000, C 0.000 }
gfCNCPoint1[13068] = {X 317.9435, Y 98.8535, Z -1.3333, A 0.000, B 0.000, C 0.000 }
gfCNCPoint1[13069] = {X 316.4423, Y 98.1619, Z -1.3333, A 0.000, B 0.000, C 0.000 }
gfCNCPoint1[13070] = {X 315.0044, Y 97.3467, Z -1.3333, A 0.000, B 0.000, C 0.000 }
gfCNCPoint1[13071] = {X 313.6400, Y 96.4139, Z -1.3333, A 0.000, B 0.000, C 0.000 }
gfCNCPoint1[13072] = {X 312.3586, Y 95.3698, Z -1.3333, A 0.000, B 0.000, C 0.000 }
gfCNCPoint1[13073] = {X 311.3689, Y 94.3848, Z -1.3333, A 0.000, B 0.000, C 0.000 }
gfCNCPoint1[13074] = {X 310.5028, Y 93.2894, Z -1.3333, A 0.000, B 0.000, C 0.000 }
gfCNCPoint1[13075] = {X 309.7726, Y 92.0992, Z -1.3333, A 0.000, B 0.000, C 0.000 }
gfCNCPoint1[13076] = {X 309.1885, Y 90.8309, Z -1.3333, A 0.000, B 0.000, C 0.000 }
gfCNCPoint1[13077] = {X 308.7589, Y 89.5022, Z -1.3333, A 0.000, B 0.000, C 0.000 }
gfCNCPoint1[13078] = {X 308.4183, Y 87.8925, Z -1.3333, A 0.000, B 0.000, C 0.000 }
gfCNCPoint1[13079] = {X 308.2170, Y 86.2594, Z -1.3333, A 0.000, B 0.000, C 0.000 }
gfCNCPoint1[13080] = {X 308.1567, Y 84.6152, Z -1.3333, A 0.000, B 0.000, C 0.000 }
gfCNCPoint1[13081] = {X 308.1580, Y 83.2311, Z -1.3333, A 0.000, B 0.000, C 0.000 }
gfCNCPoint1[13082] = {X 308.1580, Y 63.0709, Z -1.3333, A 0.000, B 0.000, C 0.000 }
gfCNCPoint1[13083] = {X 307.3126, Y 62.8911, Z -1.3333, A 0.000, B 0.000, C 0.000 }
gfCNCPoint1[13084] = {X 306.5227, Y 62.5404, Z -1.3333, A 0.000, B 0.000, C 0.000 }
gfCNCPoint1[13085] = {X 305.8222, Y 62.0341, Z -1.3333, A 0.000, B 0.000, C 0.000 }
gfCNCPoint1[13086] = {X 305.2415, Y 61.3940, Z -1.3333, A 0.000, B 0.000, C 0.000 }
gfCNCPoint1[13087] = {X 304.8056, Y 60.6477, Z -1.3333, A 0.000, B 0.000, C 0.000 }
gfCNCPoint1[13088] = {X 304.5333, Y 59.8274, Z -1.3333, A 0.000, B 0.000, C 0.000 }
gfCNCPoint1[13089] = {X 304.4364, Y 58.9686, Z -1.3333, A 0.000, B 0.000, C 0.000 }
gfCNCPoint1[13090] = {X 304.4362, Y 58.0000, Z -1.3333, A 0.000, B 0.000, C 0.000 }
gfCNCPoint1[13091] = {X 304.5405, Y 57.0743, Z -1.3333, A 0.000, B 0.000, C 0.000 }
gfCNCPoint1[13092] = {X 304.8482, Y 56.1950, Z -1.3333, A 0.000, B 0.000, C 0.000 }
gfCNCPoint1[13093] = {X 305.3438, Y 55.4063, Z -1.3333, A 0.000, B 0.000, C 0.000 }
gfCNCPoint1[13094] = {X 306.0025, Y 54.7476, Z -1.3333, A 0.000, B 0.000, C 0.000 }
gfCNCPoint1[13095] = {X 306.7913, Y 54.2520, Z -1.3333, A 0.000, B 0.000, C 0.000 }
gfCNCPoint1[13096] = {X 307.6705, Y 53.9443, Z -1.3333, A 0.000, B 0.000, C 0.000 }
gfCNCPoint1[13097] = {X 308.5962, Y 53.8400, Z -1.3333, A 0.000, B 0.000, C 0.000 }
gfCNCPoint1[13098] = {X 324.3107, Y 53.8400, Z -1.3333, A 0.000, B 0.000, C 0.000 }
gfCNCPoint1[13099] = {X 325.2364, Y 53.9443, Z -1.3333, A 0.000, B 0.000, C 0.000 }
gfCNCPoint1[13100] = {X 326.1156, Y 54.2520, Z -1.3333, A 0.000, B 0.000, C 0.000 }
gfCNCPoint1[13101] = {X 326.9044, Y 54.7476, Z -1.3333, A 0.000, B 0.000, C 0.000 }
gfCNCPoint1[13102] = {X 327.5631, Y 55.4063, Z -1.3333, A 0.000, B 0.000, C 0.000 }
gfCNCPoint1[13103] = {X 328.0587, Y 56.1950, Z -1.3333, A 0.000, B 0.000, C 0.000 }
gfCNCPoint1[13104] = {X 328.3664, Y 57.0743, Z -1.3333, A 0.000, B 0.000, C 0.000 }
gfCNCPoint1[13105] = {X 328.4707, Y 58.0000, Z -1.3333, A 0.000, B 0.000, C 0.000 }
gfCNCPoint1[13106] = {X 328.4707, Y 58.9351, Z -1.3333, A 0.000, B 0.000, C 0.000 }
gfCNCPoint1[13107] = {X 328.3755, Y 59.7983, Z -1.3333, A 0.000, B 0.000, C 0.000 }
gfCNCPoint1[13108] = {X 328.1047, Y 60.6235, Z -1.3333, A 0.000, B 0.000, C 0.000 }
gfCNCPoint1[13109] = {X 327.6701, Y 61.3753, Z -1.3333, A 0.000, B 0.000, C 0.000 }
gfCNCPoint1[13110] = {X 327.0901, Y 62.0217, Z -1.3333, A 0.000, B 0.000, C 0.000 }
gfCNCPoint1[13111] = {X 326.3895, Y 62.5350, Z -1.3333, A 0.000, B 0.000, C 0.000 }
gfCNCPoint1[13112] = {X 325.5984, Y 62.8933, Z -1.3333, A 0.000, B 0.000, C 0.000 }
gfCNCPoint1[13113] = {X 324.7505, Y 63.0811, Z -1.3333, A 0.000, B 0.000, C 0.000 }
gfCNCPoint1[13114] = {X 324.7519, Y 83.2304, Z -1.3333, A 0.000, B 0.000, C 0.000 }
gfCNCPoint1[13115] = {X 324.7654, Y 84.6154, Z -1.3333, A 0.000, B 0.000, C 0.000 }
gfCNCPoint1[13116] = {X 324.8458, Y 85.8846, Z -1.3333, A 0.000, B 0.000, C 0.000 }
gfCNCPoint1[13117] = {X 325.0778, Y 87.1350, Z -1.3333, A 0.000, B 0.000, C 0.000 }
gfCNCPoint1[13118] = {X 325.3538, Y 87.4467, Z -1.3333, A 0.000, B 0.000, C 0.000 }
gfCNCPoint1[13119] = {X 325.6979, Y 87.6811, Z -1.3333, A 0.000, B 0.000, C 0.000 }
gfCNCPoint1[13120] = {X 326.1491, Y 87.9356, Z -1.3333, A 0.000, B 0.000, C 0.000 }
gfCNCPoint1[13121] = {X 327.6059, Y 88.5415, Z -1.3333, A 0.000, B 0.000, C 0.000 }
gfCNCPoint1[13122] = {X 329.1206, Y 88.9832, Z -1.3333, A 0.000, B 0.000, C 0.000 }
gfCNCPoint1[13123] = {X 332.2075, Y 89.6012, Z -1.3333, A 0.000, B 0.000, C 0.000 }
gfCNCPoint1[13124] = {X 335.3309, Y 89.9948, Z -1.3333, A 0.000, B 0.000, C 0.000 }
gfCNCPoint1[13125] = {X 340.5120, Y 90.3783, Z -1.3333, A 0.000, B 0.000, C 0.000 }
gfCNCPoint1[13126] = {X 345.7053, Y 90.5232, Z -1.3333, A 0.000, B 0.000, C 0.000 }
gfCNCPoint1[13127] = {X 350.5525, Y 90.5292, Z -1.3333, A 0.000, B 0.000, C 0.000 }
gfCNCPoint1[13128] = {X 355.3968, Y 90.3605, Z -1.3333, A 0.000, B 0.000, C 0.000 }
gfCNCPoint1[13129] = {X 360.2319, Y 90.0174, Z -1.3333, A 0.000, B 0.000, C 0.000 }
gfCNCPoint1[13130] = {X 362.7884, Y 89.7271, Z -1.3333, A 0.000, B 0.000, C 0.000 }
gfCNCPoint1[13131] = {X 365.3213, Y 89.2752, Z -1.3333, A 0.000, B 0.000, C 0.000 }
gfCNCPoint1[13132] = {X 367.8205, Y 88.6637, Z -1.3333, A 0.000, B 0.000, C 0.000 }
gfCNCPoint1[13133] = {X 368.7693, Y 88.3446, Z -1.3333, A 0.000, B 0.000, C 0.000 }
gfCNCPoint1[13134] = {X 369.6764, Y 87.9211, Z -1.3333, A 0.000, B 0.000, C 0.000 }
gfCNCPoint1[13135] = {X 370.5302, Y 87.3986, Z -1.3333, A 0.000, B 0.000, C 0.000 }
gfCNCPoint1[13136] = {X 370.7243, Y 87.1966, Z -1.3333, A 0.000, B 0.000, C 0.000 }
gfCNCPoint1[13137] = {X 370.8244, Y 86.9349, Z -1.3333, A 0.000, B 0.000, C 0.000 }
gfCNCPoint1[13138] = {X 371.0171, Y 85.3866, Z -1.3333, A 0.000, B 0.000, C 0.000 }
gfCNCPoint1[13139] = {X 371.0814, Y 83.8276, Z -1.3333, A 0.000, B 0.000, C 0.000 }
gfCNCPoint1[13140] = {X 371.0811, Y 63.0709, Z -1.3333, A 0.000, B 0.000, C 0.000 }
gfCNCPoint1[13141] = {X 370.9788, Y 63.0588, Z -1.3333, A 0.000, B 0.000, C 0.000 }
gfCNCPoint1[13142] = {X 370.8767, Y 63.0441, Z -1.3333, A 0.000, B 0.000, C 0.000 }
gfCNCPoint1[13143] = {X 369.9390, Y 62.7822, Z -1.3333, A 0.000, B 0.000, C 0.000 }
gfCNCPoint1[13144] = {X 369.0879, Y 62.3095, Z -1.3333, A 0.000, B 0.000, C 0.000 }
gfCNCPoint1[13145] = {X 368.3699, Y 61.6520, Z -1.3333, A 0.000, B 0.000, C 0.000 }
gfCNCPoint1[13146] = {X 367.8244, Y 60.8455, Z -1.3333, A 0.000, B 0.000, C 0.000 }
gfCNCPoint1[13147] = {X 367.4813, Y 59.9344, Z -1.3333, A 0.000, B 0.000, C 0.000 }
gfCNCPoint1[13148] = {X 367.3594, Y 58.9684, Z -1.3333, A 0.000, B 0.000, C 0.000 }
gfCNCPoint1[13149] = {X 367.3593, Y 58.0000, Z -1.3333, A 0.000, B 0.000, C 0.000 }
gfCNCPoint1[13150] = {X 367.4636, Y 57.0743, Z -1.3333, A 0.000, B 0.000, C 0.000 }
gfCNCPoint1[13151] = {X 367.7713, Y 56.1950, Z -1.3333, A 0.000, B 0.000, C 0.000 }
gfCNCPoint1[13152] = {X 368.2669, Y 55.4063, Z -1.3333, A 0.000, B 0.000, C 0.000 }
gfCNCPoint1[13153] = {X 368.9256, Y 54.7476, Z -1.3333, A 0.000, B 0.000, C 0.000 }
gfCNCPoint1[13154] = {X 369.7143, Y 54.2520, Z -1.3333, A 0.000, B 0.000, C 0.000 }
gfCNCPoint1[13155] = {X 370.5936, Y 53.9443, Z -1.3333, A 0.000, B 0.000, C 0.000 }
gfCNCPoint1[13156] = {X 371.5193, Y 53.8400, Z -1.3333, A 0.000, B 0.000, C 0.000 }
gfCNCPoint1[13157] = {X 388.0597, Y 53.8400, Z -1.3333, A 0.000, B 0.000, C 0.000 }
gfCNCPoint1[13158] = {X 388.9854, Y 53.9443, Z -1.3333, A 0.000, B 0.000, C 0.000 }
gfCNCPoint1[13159] = {X 389.8646, Y 54.2520, Z -1.3333, A 0.000, B 0.000, C 0.000 }
gfCNCPoint1[13160] = {X 390.6534, Y 54.7476, Z -1.3333, A 0.000, B 0.000, C 0.000 }
gfCNCPoint1[13161] = {X 391.3121, Y 55.4063, Z -1.3333, A 0.000, B 0.000, C 0.000 }
gfCNCPoint1[13162] = {X 391.8077, Y 56.1950, Z -1.3333, A 0.000, B 0.000, C 0.000 }
gfCNCPoint1[13163] = {X 392.1154, Y 57.0743, Z -1.3333, A 0.000, B 0.000, C 0.000 }
gfCNCPoint1[13164] = {X 392.2197, Y 58.0000, Z -1.3333, A 0.000, B 0.000, C 0.000 }
gfCNCPoint1[13165] = {X 392.2197, Y 58.9342, Z -1.3333, A 0.000, B 0.000, C 0.000 }
gfCNCPoint1[13166] = {X 392.1077, Y 59.8928, Z -1.3333, A 0.000, B 0.000, C 0.000 }
gfCNCPoint1[13167] = {X 391.7778, Y 60.7998, Z -1.3333, A 0.000, B 0.000, C 0.000 }
gfCNCPoint1[13168] = {X 391.2335, Y 61.6243, Z -1.3333, A 0.000, B 0.000, C 0.000 }
gfCNCPoint1[13169] = {X 390.5109, Y 62.2980, Z -1.3333, A 0.000, B 0.000, C 0.000 }
gfCNCPoint1[13170] = {X 389.6503, Y 62.7834, Z -1.3333, A 0.000, B 0.000, C 0.000 }
gfCNCPoint1[13171] = {X 388.6998, Y 63.0532, Z -1.3333, A 0.000, B 0.000, C 0.000 }
gfCNCPoint1[13172] = {X 388.5996, Y 63.0679, Z -1.3333, A 0.000, B 0.000, C 0.000 }
gfCNCPoint1[13173] = {X 388.4990, Y 63.0803, Z -1.3333, A 0.000, B 0.000, C 0.000 }
gfCNCPoint1[13174] = {X 388.4956, Y 84.6154, Z -1.3333, A 0.000, B 0.000, C 0.000 }
gfCNCPoint1[13175] = {X 388.4361, Y 86.2600, Z -1.3333, A 0.000, B 0.000, C 0.000 }
gfCNCPoint1[13176] = {X 388.2335, Y 87.8931, Z -1.3333, A 0.000, B 0.000, C 0.000 }
gfCNCPoint1[13177] = {X 387.8893, Y 89.5024, Z -1.3333, A 0.000, B 0.000, C 0.000 }
gfCNCPoint1[13178] = {X 387.3644, Y 91.0684, Z -1.3333, A 0.000, B 0.000, C 0.000 }
gfCNCPoint1[13179] = {X 386.6250, Y 92.5454, Z -1.3333, A 0.000, B 0.000, C 0.000 }
gfCNCPoint1[13180] = {X 385.6856, Y 93.9039, Z -1.3333, A 0.000, B 0.000, C 0.000 }
gfCNCPoint1[13181] = {X 384.5649, Y 95.1172, Z -1.3333, A 0.000, B 0.000, C 0.000 }
gfCNCPoint1[13182] = {X 383.0638, Y 96.3817, Z -1.3333, A 0.000, B 0.000, C 0.000 }
gfCNCPoint1[13183] = {X 381.4371, Y 97.4797, Z -1.3333, A 0.000, B 0.000, C 0.000 }
gfCNCPoint1[13184] = {X 379.7031, Y 98.3990, Z -1.3333, A 0.000, B 0.000, C 0.000 }
gfCNCPoint1[13185] = {X 377.4429, Y 99.3519, Z -1.3333, A 0.000, B 0.000, C 0.000 }
gfCNCPoint1[13186] = {X 375.1196, Y 100.1385, Z -1.3333, A 0.000, B 0.000, C 0.000 }
gfCNCPoint1[13187] = {X 372.7454, Y 100.7548, Z -1.3333, A 0.000, B 0.000, C 0.000 }
gfCNCPoint1[13188] = {X 368.9414, Y 101.4907, Z -1.3333, A 0.000, B 0.000, C 0.000 }
gfCNCPoint1[13189] = {X 365.1065, Y 102.0429, Z -1.3333, A 0.000, B 0.000, C 0.000 }
gfCNCPoint1[13190] = {X 361.2495, Y 102.4101, Z -1.3333, A 0.000, B 0.000, C 0.000 }
gfCNCPoint1[13191] = {X 357.2460, Y 102.6506, Z -1.3333, A 0.000, B 0.000, C 0.000 }
gfCNCPoint1[13192] = {X 353.2382, Y 102.8039, Z -1.3333, A 0.000, B 0.000, C 0.000 }
gfCNCPoint1[13193] = {X 353.3477, Y 106.8024, Z -1.3333, A 0.000, B 0.000, C 0.000 }
gfCNCPoint1[13194] = {X 353.2361, Y 102.7240, Z -1.3333, A 0.000, B 0.000, C 0.000 }
gfCNCPoint1[13195] = {X 347.7209, Y 102.7924, Z -1.3333, A 0.000, B 0.000, C 0.000 }
gfCNCPoint1[13196] = {X 342.2061, Y 102.6958, Z -1.3333, A 0.000, B 0.000, C 0.000 }
gfCNCPoint1[13197] = {X 336.6968, Y 102.4342, Z -1.3333, A 0.000, B 0.000, C 0.000 }
gfCNCPoint1[13198] = {X 333.2159, Y 102.1599, Z -1.3333, A 0.000, B 0.000, C 0.000 }
gfCNCPoint1[13199] = {X 329.7487, Y 101.7481, Z -1.3333, A 0.000, B 0.000, C 0.000 }
gfCNCPoint1[13200] = {X 326.3005, Y 101.1993, Z -1.3333, A 0.000, B 0.000, C 0.000 }
gfCNCPoint1[13201] = {X 323.4679, Y 100.5985, Z -1.3333, A 0.000, B 0.000, C 0.000 }
gfCNCPoint1[13202] = {X 320.6874, Y 99.7904, Z -1.3333, A 0.000, B 0.000, C 0.000 }
gfCNCPoint1[13203] = {X 317.9740, Y 98.7795, Z -1.3333, A 0.000, B 0.000, C 0.000 }
gfCNCPoint1[13204] = {X 316.4789, Y 98.0907, Z -1.3333, A 0.000, B 0.000, C 0.000 }
gfCNCPoint1[13205] = {X 315.0468, Y 97.2789, Z -1.3333, A 0.000, B 0.000, C 0.000 }
gfCNCPoint1[13206] = {X 313.6879, Y 96.3498, Z -1.3333, A 0.000, B 0.000, C 0.000 }
gfCNCPoint1[13207] = {X 312.4117, Y 95.3100, Z -1.3333, A 0.000, B 0.000, C 0.000 }
gfCNCPoint1[13208] = {X 311.4286, Y 94.3316, Z -1.3333, A 0.000, B 0.000, C 0.000 }
gfCNCPoint1[13209] = {X 310.5684, Y 93.2437, Z -1.3333, A 0.000, B 0.000, C 0.000 }
gfCNCPoint1[13210] = {X 309.8432, Y 92.0616, Z -1.3333, A 0.000, B 0.000, C 0.000 }
gfCNCPoint1[13211] = {X 309.2631, Y 90.8018, Z -1.3333, A 0.000, B 0.000, C 0.000 }
gfCNCPoint1[13212] = {X 308.8363, Y 89.4822, Z -1.3333, A 0.000, B 0.000, C 0.000 }
gfCNCPoint1[13213] = {X 308.4971, Y 87.8792, Z -1.3333, A 0.000, B 0.000, C 0.000 }
gfCNCPoint1[13214] = {X 308.2968, Y 86.2529, Z -1.3333, A 0.000, B 0.000, C 0.000 }
gfCNCPoint1[13215] = {X 308.2367, Y 84.6155, Z -1.3333, A 0.000, B 0.000, C 0.000 }
gfCNCPoint1[13216] = {X 308.2380, Y 83.2312, Z -1.3333, A 0.000, B 0.000, C 0.000 }
gfCNCPoint1[13217] = {X 308.2380, Y 62.9983, Z -1.3333, A 0.000, B 0.000, C 0.000 }
gfCNCPoint1[13218] = {X 307.3961, Y 62.8336, Z -1.3333, A 0.000, B 0.000, C 0.000 }
gfCNCPoint1[13219] = {X 306.6072, Y 62.4964, Z -1.3333, A 0.000, B 0.000, C 0.000 }
gfCNCPoint1[13220] = {X 305.9063, Y 62.0018, Z -1.3333, A 0.000, B 0.000, C 0.000 }
gfCNCPoint1[13221] = {X 305.3243, Y 61.3715, Z -1.3333, A 0.000, B 0.000, C 0.000 }
gfCNCPoint1[13222] = {X 304.8870, Y 60.6335, Z -1.3333, A 0.000, B 0.000, C 0.000 }
gfCNCPoint1[13223] = {X 304.6136, Y 59.8203, Z -1.3333, A 0.000, B 0.000, C 0.000 }
gfCNCPoint1[13224] = {X 304.5164, Y 58.9680, Z -1.3333, A 0.000, B 0.000, C 0.000 }
gfCNCPoint1[13225] = {X 304.5162, Y 58.0000, Z -1.3333, A 0.000, B 0.000, C 0.000 }
gfCNCPoint1[13226] = {X 304.6185, Y 57.0921, Z -1.3333, A 0.000, B 0.000, C 0.000 }
gfCNCPoint1[13227] = {X 304.9203, Y 56.2298, Z -1.3333, A 0.000, B 0.000, C 0.000 }
gfCNCPoint1[13228] = {X 305.4064, Y 55.4562, Z -1.3333, A 0.000, B 0.000, C 0.000 }
gfCNCPoint1[13229] = {X 306.0524, Y 54.8101, Z -1.3333, A 0.000, B 0.000, C 0.000 }
gfCNCPoint1[13230] = {X 306.8260, Y 54.3240, Z -1.3333, A 0.000, B 0.000, C 0.000 }
gfCNCPoint1[13231] = {X 307.6883, Y 54.0223, Z -1.3333, A 0.000, B 0.000, C 0.000 }
gfCNCPoint1[13232] = {X 308.5962, Y 53.9200, Z -1.3333, A 0.000, B 0.000, C 0.000 }
gfCNCPoint1[13233] = {X 324.3107, Y 53.9200, Z -1.3333, A 0.000, B 0.000, C 0.000 }
gfCNCPoint1[13234] = {X 325.2186, Y 54.0223, Z -1.3333, A 0.000, B 0.000, C 0.000 }
gfCNCPoint1[13235] = {X 326.0809, Y 54.3240, Z -1.3333, A 0.000, B 0.000, C 0.000 }
gfCNCPoint1[13236] = {X 326.8545, Y 54.8101, Z -1.3333, A 0.000, B 0.000, C 0.000 }
gfCNCPoint1[13237] = {X 327.5006, Y 55.4562, Z -1.3333, A 0.000, B 0.000, C 0.000 }
gfCNCPoint1[13238] = {X 327.9866, Y 56.2298, Z -1.3333, A 0.000, B 0.000, C 0.000 }
gfCNCPoint1[13239] = {X 328.2884, Y 57.0921, Z -1.3333, A 0.000, B 0.000, C 0.000 }
gfCNCPoint1[13240] = {X 328.3907, Y 58.0000, Z -1.3333, A 0.000, B 0.000, C 0.000 }
gfCNCPoint1[13241] = {X 328.3907, Y 58.9346, Z -1.3333, A 0.000, B 0.000, C 0.000 }
gfCNCPoint1[13242] = {X 328.2951, Y 59.7913, Z -1.3333, A 0.000, B 0.000, C 0.000 }
gfCNCPoint1[13243] = {X 328.0233, Y 60.6094, Z -1.3333, A 0.000, B 0.000, C 0.000 }
gfCNCPoint1[13244] = {X 327.5873, Y 61.3530, Z -1.3333, A 0.000, B 0.000, C 0.000 }
gfCNCPoint1[13245] = {X 327.0061, Y 61.9896, Z -1.3333, A 0.000, B 0.000, C 0.000 }
gfCNCPoint1[13246] = {X 326.3051, Y 62.4914, Z -1.3333, A 0.000, B 0.000, C 0.000 }
gfCNCPoint1[13247] = {X 325.5150, Y 62.8362, Z -1.3333, A 0.000, B 0.000, C 0.000 }
gfCNCPoint1[13248] = {X 324.6705, Y 63.0092, Z -1.3333, A 0.000, B 0.000, C 0.000 }
gfCNCPoint1[13249] = {X 324.6719, Y 83.2309, Z -1.3333, A 0.000, B 0.000, C 0.000 }
gfCNCPoint1[13250] = {X 324.6854, Y 84.6157, Z -1.3333, A 0.000, B 0.000, C 0.000 }
gfCNCPoint1[13251] = {X 324.7673, Y 85.9016, Z -1.3333, A 0.000, B 0.000, C 0.000 }
gfCNCPoint1[13252] = {X 325.0037, Y 87.1682, Z -1.3333, A 0.000, B 0.000, C 0.000 }
gfCNCPoint1[13253] = {X 325.2949, Y 87.5014, Z -1.3333, A 0.000, B 0.000, C 0.000 }
gfCNCPoint1[13254] = {X 325.6599, Y 87.7516, Z -1.3333, A 0.000, B 0.000, C 0.000 }
gfCNCPoint1[13255] = {X 326.1120, Y 88.0066, Z -1.3333, A 0.000, B 0.000, C 0.000 }
gfCNCPoint1[13256] = {X 327.5781, Y 88.6166, Z -1.3333, A 0.000, B 0.000, C 0.000 }
gfCNCPoint1[13257] = {X 329.1024, Y 89.0611, Z -1.3333, A 0.000, B 0.000, C 0.000 }
gfCNCPoint1[13258] = {X 332.1948, Y 89.6802, Z -1.3333, A 0.000, B 0.000, C 0.000 }
gfCNCPoint1[13259] = {X 335.3238, Y 90.0745, Z -1.3333, A 0.000, B 0.000, C 0.000 }
gfCNCPoint1[13260] = {X 340.5083, Y 90.4582, Z -1.3333, A 0.000, B 0.000, C 0.000 }
gfCNCPoint1[13261] = {X 345.7049, Y 90.6032, Z -1.3333, A 0.000, B 0.000, C 0.000 }
gfCNCPoint1[13262] = {X 350.5546, Y 90.6091, Z -1.3333, A 0.000, B 0.000, C 0.000 }
gfCNCPoint1[13263] = {X 355.4014, Y 90.4404, Z -1.3333, A 0.000, B 0.000, C 0.000 }
gfCNCPoint1[13264] = {X 360.2390, Y 90.0971, Z -1.3333, A 0.000, B 0.000, C 0.000 }
gfCNCPoint1[13265] = {X 362.8003, Y 89.8062, Z -1.3333, A 0.000, B 0.000, C 0.000 }
gfCNCPoint1[13266] = {X 365.3380, Y 89.3534, Z -1.3333, A 0.000, B 0.000, C 0.000 }
